LIN {X 0,Y 240.395,Z 425.258,A -85,B 0,C 180,E1 -19814.358,E2 -19814.358} C_VEL
LIN {X 0,Y 237.821,Z 422.9,A -85,B 0,C 180,E1 -19816.141,E2 -19816.141} C_VEL
LIN {X 0,Y 236.639,Z 420.217,A -85,B 0,C 180,E1 -19817.343,E2 -19817.343} C_VEL
LIN {X 0,Y 236.604,Z 420.167,A -85,B 0,C 180,E1 -19820.883,E2 -19820.883} C_VEL
LIN {X 0,Y 236.627,Z 420.436,A -85,B 0,C 180,E1 -19824.572,E2 -19824.572} C_VEL
LIN {X 0,Y 236.725,Z 421.066,A -85,B 0,C 180,E1 -19828.362,E2 -19828.362} C_VEL
LIN {X 0,Y 236.86,Z 422.112,A -85,B 0,C 180,E1 -19832.284,E2 -19832.284} C_VEL
LIN {X 0,Y 237.127,Z 423.615,A -85,B 0,C 180,E1 -19836.355,E2 -19836.355} C_VEL
LIN {X 0,Y 237.519,Z 425.71,A -85,B 0,C 180,E1 -19840.616,E2 -19840.616} C_VEL
LIN {X 0,Y 237.77,Z 427.097,A -85,B 0,C 180,E1 -19843.015,E2 -19843.015} C_VEL
LIN {X 0,Y 237.655,Z 428.197,A -85,B 0,C 180,E1 -19843.759,E2 -19843.759} C_VEL
LIN {X 0,Y 237.217,Z 431.036,A -85,B 0,C 180,E1 -19844.653,E2 -19844.653} C_VEL
LIN {X 0,Y 236.854,Z 438.007,A -85,B 0,C 180,E1 -19846.253,E2 -19846.253} C_VEL
LIN {X 0,Y 237.602,Z 440.293,A -85,B 0,C 180,E1 -19847.045,E2 -19847.045} C_VEL
LIN {X 0,Y 238.71,Z 442.196,A -85,B 0,C 180,E1 -19847.865,E2 -19847.865} C_VEL
LIN {X 0,Y 241.116,Z 447.739,A -85,B 0,C 180,E1 -19849.805,E2 -19849.805} C_VEL
LIN {X 0,Y 243.272,Z 454.639,A -85,B 0,C 180,E1 -19851.771,E2 -19851.771} C_VEL
LIN {X 0,Y 245.138,Z 466.004,A -85,B 0,C 180,E1 -19854.44,E2 -19854.44} C_VEL
LIN {X 0,Y 245.966,Z 476.957,A -85,B 0,C 180,E1 -19856.903,E2 -19856.903} C_VEL
LIN {X 0,Y 245.658,Z 486.508,A -85,B 0,C 180,E1 -19859.013,E2 -19859.013} C_VEL
LIN {X 0,Y 244.271,Z 496.15,A -85,B 0,C 180,E1 -19861.197,E2 -19861.197} C_VEL
LIN {X 0,Y 242.996,Z 501.368,A -85,B 0,C 180,E1 -19862.443,E2 -19862.443} C_VEL
LIN {X 0,Y 239.073,Z 510.716,A -85,B 0,C 180,E1 -19864.778,E2 -19864.778} C_VEL
LIN {X 0,Y 235.521,Z 518.441,A -85,B 0,C 180,E1 -19867.182,E2 -19867.182} C_VEL
LIN {X 0,Y 232.602,Z 524.845,A -85,B 0,C 180,E1 -19869.702,E2 -19869.702} C_VEL
LIN {X 0,Y 230.441,Z 529.963,A -85,B 0,C 180,E1 -19872.25,E2 -19872.25} C_VEL
LIN {X 0,Y 227.887,Z 535.233,A -85,B 0,C 180,E1 -19875.724,E2 -19875.724} C_VEL
LIN {X 0,Y 227.074,Z 537.27,A -85,B 0,C 180,E1 -19877.495,E2 -19877.495} C_VEL
LIN {X 0,Y 226.494,Z 538.88,A -85,B 0,C 180,E1 -19879.277,E2 -19879.277} C_VEL
LIN {X 0,Y 225.828,Z 540.91,A -85,B 0,C 180,E1 -19882.856,E2 -19882.856} C_VEL
LIN {X 0,Y 225.781,Z 541.415,A -85,B 0,C 180,E1 -19884.939,E2 -19884.939} C_VEL
LIN {X 0,Y 225.916,Z 541.064,A -85,B 0,C 180,E1 -19888.224,E2 -19888.224} C_VEL
LIN {X 0,Y 226.064,Z 540.289,A -85,B 0,C 180,E1 -19890.007,E2 -19890.007} C_VEL
LIN {X 0,Y 225.977,Z 539.082,A -85,B 0,C 180,E1 -19891.789,E2 -19891.789} C_VEL
LIN {X 0,Y 226.017,Z 536.428,A -85,B 0,C 180,E1 -19894.465,E2 -19894.465} C_VEL
LIN {X 0,Y 226.071,Z 532.684,A -85,B 0,C 180,E1 -19897.15,E2 -19897.15} C_VEL
LIN {X 0,Y 226.387,Z 527.772,A -85,B 0,C 180,E1 -19899.837,E2 -19899.837} C_VEL
LIN {X 0,Y 227.006,Z 521.552,A -85,B 0,C 180,E1 -19902.523,E2 -19902.523} C_VEL
LIN {X 0,Y 228.165,Z 513.778,A -85,B 0,C 180,E1 -19905.184,E2 -19905.184} C_VEL
LIN {X 0,Y 229.487,Z 504.066,A -85,B 0,C 180,E1 -19907.839,E2 -19907.839} C_VEL
LIN {X 0,Y 231.269,Z 494.144,A -85,B 0,C 180,E1 -19909.997,E2 -19909.997} C_VEL
LIN {X 0,Y 232.165,Z 486.97,A -85,B 0,C 180,E1 -19911.307,E2 -19911.307} C_VEL
LIN {X 0,Y 231.576,Z 476.41,A -85,B 0,C 180,E1 -19913.007,E2 -19913.007} C_VEL
LIN {X 0,Y 230.692,Z 464.985,A -85,B 0,C 180,E1 -19914.519,E2 -19914.519} C_VEL
LIN {X 0,Y 229.348,Z 451.694,A -85,B 0,C 180,E1 -19915.93,E2 -19915.93} C_VEL
LIN {X 0,Y 227.728,Z 438.212,A -85,B 0,C 180,E1 -19917.017,E2 -19917.017} C_VEL
LIN {X 0,Y 227.566,Z 436.511,A -85,B 0,C 180,E1 -19917.125,E2 -19917.125} C_VEL
LIN {X 0,Y 228.588,Z 431.326,A -85,B 0,C 180,E1 -19921.518,E2 -19921.518} C_VEL
LIN {X 0,Y 229.756,Z 426.613,A -85,B 0,C 180,E1 -19925.541,E2 -19925.541} C_VEL
LIN {X 0,Y 230.008,Z 424.188,A -85,B 0,C 180,E1 -19927.676,E2 -19927.676} C_VEL
LIN {X 0,Y 229.5,Z 420.39,A -85,B 0,C 180,E1 -19931.183,E2 -19931.183} C_VEL
LIN {X 0,Y 228.708,Z 416.42,A -85,B 0,C 180,E1 -19935.025,E2 -19935.025} C_VEL
LIN {X 0,Y 227.915,Z 412.095,A -85,B 0,C 180,E1 -19939.495,E2 -19939.495} C_VEL
LIN {X 0,Y 227.883,Z 412.095,A -85,B 0,C 180,E1 -19944.127,E2 -19944.127} C_VEL
LIN {X 0,Y 227.875,Z 412.098,A -85,B 0,C 180,E1 -19948.377,E2 -19948.377} C_VEL
LIN {X 0,Y 227.874,Z 412.097,A -85,B 0,C 180,E1 -19952.442,E2 -19952.442} C_VEL
LIN {X 0,Y 227.909,Z 412.094,A -85,B 0,C 180,E1 -19956.365,E2 -19956.365} C_VEL
LIN {X 0,Y 227.916,Z 412.092,A -85,B 0,C 180,E1 -19960.171,E2 -19960.171} C_VEL
LIN {X 0,Y 228.037,Z 412.077,A -85,B 0,C 180,E1 -19963.895,E2 -19963.895} C_VEL
LIN {X 0,Y 228.072,Z 412.073,A -85,B 0,C 180,E1 -19967.542,E2 -19967.542} C_VEL
LIN {X 0,Y 228.276,Z 412.05,A -85,B 0,C 180,E1 -19971.143,E2 -19971.143} C_VEL
LIN {X 0,Y 228.329,Z 412.044,A -85,B 0,C 180,E1 -19972.926,E2 -19972.926} C_VEL
LIN {X 0,Y 228.568,Z 412.009,A -85,B 0,C 180,E1 -19978.236,E2 -19978.236} C_VEL
LIN {X 0,Y 228.556,Z 412.013,A -85,B 0,C 180,E1 -19981.761,E2 -19981.761} C_VEL
LIN {X 0,Y 228.315,Z 412.044,A -85,B 0,C 180,E1 -19987.071,E2 -19987.071} C_VEL
LIN {X 0,Y 228.157,Z 412.065,A -85,B 0,C 180,E1 -19990.649,E2 -19990.649} C_VEL
LIN {X 0,Y 228.047,Z 412.076,A -85,B 0,C 180,E1 -19994.272,E2 -19994.272} C_VEL
LIN {X 0,Y 227.945,Z 412.089,A -85,B 0,C 180,E1 -19997.956,E2 -19997.956} C_VEL
LIN {X 0,Y 227.914,Z 412.093,A -85,B 0,C 180,E1 -20002.306,E2 -20002.306} C_VEL
LIN {X 0,Y 227.954,Z 412.091,A -85,B 0,C 180,E1 -20006.597,E2 -20006.597} C_VEL
LIN {X 0,Y 227.89,Z 412.097,A -85,B 0,C 180,E1 -20010.278,E2 -20010.278} C_VEL
LIN {X 0,Y 227.889,Z 412.095,A -85,B 0,C 180,E1 -20013.716,E2 -20013.716} C_VEL
LIN {X 0,Y 227.855,Z 412.101,A -85,B 0,C 180,E1 -20018.087,E2 -20018.087} C_VEL
LIN {X 0,Y 227.815,Z 412.108,A -85,B 0,C 180,E1 -20022.739,E2 -20022.739} C_VEL
LIN {X 0,Y 227.811,Z 412.104,A -85,B 0,C 180,E1 -20027.25,E2 -20027.25} C_VEL
LIN {X 0,Y 227.85,Z 412.101,A -85,B 0,C 180,E1 -20031.903,E2 -20031.903} C_VEL
LIN {X 0,Y 227.885,Z 412.098,A -85,B 0,C 180,E1 -20036.372,E2 -20036.372} C_VEL
LIN {X 0,Y 227.923,Z 412.096,A -85,B 0,C 180,E1 -20040.432,E2 -20040.432} C_VEL
LIN {X 0,Y 227.932,Z 412.091,A -85,B 0,C 180,E1 -20044.42,E2 -20044.42} C_VEL
LIN {X 0,Y 227.965,Z 412.09,A -85,B 0,C 180,E1 -20048.281,E2 -20048.281} C_VEL
LIN {X 0,Y 228.035,Z 412.076,A -85,B 0,C 180,E1 -20052.82,E2 -20052.82} C_VEL
LIN {X 0,Y 228.071,Z 412.074,A -85,B 0,C 180,E1 -20057.537,E2 -20057.537} C_VEL
LIN {X 0,Y 228.265,Z 412.047,A -85,B 0,C 180,E1 -20061.138,E2 -20061.138} C_VEL
LIN {X 0,Y 228.32,Z 412.041,A -85,B 0,C 180,E1 -20062.921,E2 -20062.921} C_VEL
LIN {X 0,Y 228.548,Z 412.016,A -85,B 0,C 180,E1 -20068.231,E2 -20068.231} C_VEL
LIN {X 0,Y 228.548,Z 412.013,A -85,B 0,C 180,E1 -20071.756,E2 -20071.756} C_VEL
LIN {X 0,Y 228.348,Z 412.038,A -85,B 0,C 180,E1 -20077.065,E2 -20077.065} C_VEL
LIN {X 0,Y 228.16,Z 412.063,A -85,B 0,C 180,E1 -20080.644,E2 -20080.644} C_VEL
LIN {X 0,Y 228.044,Z 412.077,A -85,B 0,C 180,E1 -20086.096,E2 -20086.096} C_VEL
LIN {X 0,Y 227.921,Z 412.094,A -85,B 0,C 180,E1 -20089.82,E2 -20089.82} C_VEL
LIN {X 0,Y 227.835,Z 412.104,A -85,B 0,C 180,E1 -20093.633,E2 -20093.633} C_VEL
LIN {X 0,Y 227.596,Z 412.134,A -85,B 0,C 180,E1 -20097.585,E2 -20097.585} C_VEL
LIN {X 0,Y 227.351,Z 412.166,A -85,B 0,C 180,E1 -20100.058,E2 -20100.058} C_VEL
LIN {X 0,Y 226.798,Z 412.354,A -85,B 0,C 180,E1 -20105.037,E2 -20105.037} C_VEL
LIN {X 0,Y 229.937,Z 425.401,A -85,B 0,C 180,E1 -20106.238,E2 -20106.238} C_VEL
LIN {X 0,Y 232.669,Z 438.268,A -85,B 0,C 180,E1 -20107.723,E2 -20107.723} C_VEL
LIN {X 0,Y 234.88,Z 450.436,A -85,B 0,C 180,E1 -20109.443,E2 -20109.443} C_VEL
LIN {X 0,Y 233.284,Z 461.497,A -85,B 0,C 180,E1 -20111.138,E2 -20111.138} C_VEL
LIN {X 0,Y 231.588,Z 472.576,A -85,B 0,C 180,E1 -20113.256,E2 -20113.256} C_VEL
LIN {X 0,Y 229.953,Z 482.534,A -85,B 0,C 180,E1 -20115.646,E2 -20115.646} C_VEL
LIN {X 0,Y 228.635,Z 490.664,A -85,B 0,C 180,E1 -20118.045,E2 -20118.045} C_VEL
LIN {X 0,Y 227.625,Z 497.485,A -85,B 0,C 180,E1 -20120.511,E2 -20120.511} C_VEL
LIN {X 0,Y 226.877,Z 502.686,A -85,B 0,C 180,E1 -20122.813,E2 -20122.813} C_VEL
LIN {X 0,Y 226.214,Z 508.373,A -85,B 0,C 180,E1 -20126,E2 -20126} C_VEL
LIN {X 0,Y 225.792,Z 512.402,A -85,B 0,C 180,E1 -20129.1,E2 -20129.1} C_VEL
LIN {X 0,Y 225.652,Z 515.079,A -85,B 0,C 180,E1 -20132.151,E2 -20132.151} C_VEL
LIN {X 0,Y 225.873,Z 516.315,A -85,B 0,C 180,E1 -20134.447,E2 -20134.447} C_VEL
LIN {X 0,Y 226.125,Z 516.805,A -85,B 0,C 180,E1 -20136.171,E2 -20136.171} C_VEL
LIN {X 0,Y 226.703,Z 516.93,A -85,B 0,C 180,E1 -20138.417,E2 -20138.417} C_VEL
LIN {X 0,Y 227.291,Z 516.575,A -85,B 0,C 180,E1 -20140.117,E2 -20140.117} C_VEL
LIN {X 0,Y 228.369,Z 515.473,A -85,B 0,C 180,E1 -20142.529,E2 -20142.529} C_VEL
LIN {X 0,Y 230.39,Z 512.669,A -85,B 0,C 180,E1 -20145.877,E2 -20145.877} C_VEL
LIN {X 0,Y 232.621,Z 509.086,A -85,B 0,C 180,E1 -20148.676,E2 -20148.676} C_VEL
LIN {X 0,Y 235.316,Z 504.302,A -85,B 0,C 180,E1 -20151.413,E2 -20151.413} C_VEL
LIN {X 0,Y 238.496,Z 498.196,A -85,B 0,C 180,E1 -20154.082,E2 -20154.082} C_VEL
LIN {X 0,Y 242.228,Z 490.525,A -85,B 0,C 180,E1 -20156.675,E2 -20156.675} C_VEL
LIN {X 0,Y 245.987,Z 481.918,A -85,B 0,C 180,E1 -20158.951,E2 -20158.951} C_VEL
LIN {X 0,Y 249.82,Z 472.11,A -85,B 0,C 180,E1 -20161.009,E2 -20161.009} C_VEL
LIN {X 0,Y 250.157,Z 471.048,A -85,B 0,C 180,E1 -20161.209,E2 -20161.209} C_VEL
LIN {X 0,Y 250.135,Z 467.345,A -85,B 0,C 180,E1 -20162.198,E2 -20162.198} C_VEL
LIN {X 0,Y 248.511,Z 456.289,A -85,B 0,C 180,E1 -20165.275,E2 -20165.275} C_VEL
LIN {X 0,Y 247.07,Z 450.957,A -85,B 0,C 180,E1 -20166.903,E2 -20166.903} C_VEL
LIN {X 0,Y 243.973,Z 443.043,A -85,B 0,C 180,E1 -20169.59,E2 -20169.59} C_VEL
LIN {X 0,Y 240.468,Z 436.403,A -85,B 0,C 180,E1 -20172.332,E2 -20172.332} C_VEL
LIN {X 0,Y 238.036,Z 432.974,A -85,B 0,C 180,E1 -20174.155,E2 -20174.155} C_VEL
LIN {X 0,Y 237.523,Z 431.74,A -85,B 0,C 180,E1 -20174.656,E2 -20174.656} C_VEL
LIN {X 0,Y 234.864,Z 428.845,A -85,B 0,C 180,E1 -20176.781,E2 -20176.781} C_VEL
LIN {X 0,Y 233.933,Z 426.768,A -85,B 0,C 180,E1 -20177.799,E2 -20177.799} C_VEL
LIN {X 0,Y 231.195,Z 424.804,A -85,B 0,C 180,E1 -20180.37,E2 -20180.37} C_VEL
LIN {X 0,Y 229.79,Z 422.242,A -85,B 0,C 180,E1 -20182.459,E2 -20182.459} C_VEL
LIN {X 0,Y 229.723,Z 421.918,A -85,B 0,C 180,E1 -20182.783,E2 -20182.783} C_VEL
LIN {X 0,Y 229.799,Z 422.557,A -85,B 0,C 180,E1 -20187.53,E2 -20187.53} C_VEL
LIN {X 0,Y 229.913,Z 423.479,A -85,B 0,C 180,E1 -20191.311,E2 -20191.311} C_VEL
LIN {X 0,Y 230.131,Z 424.91,A -85,B 0,C 180,E1 -20195.469,E2 -20195.469} C_VEL
LIN {X 0,Y 230.549,Z 426.955,A -85,B 0,C 180,E1 -20199.983,E2 -20199.983} C_VEL
LIN {X 0,Y 230.78,Z 427.896,A -85,B 0,C 180,E1 -20200.528,E2 -20200.528} C_VEL
LIN {X 0,Y 232.478,Z 431.639,A -85,B 0,C 180,E1 -20202.592,E2 -20202.592} C_VEL
LIN {X 0,Y 235.284,Z 435.262,A -85,B 0,C 180,E1 -20204.981,E2 -20204.981} C_VEL
LIN {X 0,Y 236.767,Z 439.078,A -85,B 0,C 180,E1 -20206.443,E2 -20206.443} C_VEL
LIN {X 0,Y 237.602,Z 440.293,A -85,B 0,C 180,E1 -20207.045,E2 -20207.045} C_VEL
LIN {X 0,Y 238.57,Z 442.303,A -85,B 0,C 180,E1 -20207.821,E2 -20207.821} C_VEL
LIN {X 0,Y 239.346,Z 446.289,A -85,B 0,C 180,E1 -20208.853,E2 -20208.853} C_VEL
LIN {X 0,Y 239.528,Z 450.901,A -85,B 0,C 180,E1 -20209.76,E2 -20209.76} C_VEL
LIN {X 0,Y 239.223,Z 460.716,A -85,B 0,C 180,E1 -20211.548,E2 -20211.548} C_VEL
LIN {X 0,Y 239.322,Z 463.717,A -85,B 0,C 180,E1 -20212.216,E2 -20212.216} C_VEL
LIN {X 0,Y 240.312,Z 474.933,A -85,B 0,C 180,E1 -20214.974,E2 -20214.974} C_VEL
LIN {X 0,Y 240.144,Z 484.437,A -85,B 0,C 180,E1 -20217.228,E2 -20217.228} C_VEL
LIN {X 0,Y 238.986,Z 493.867,A -85,B 0,C 180,E1 -20219.474,E2 -20219.474} C_VEL
LIN {X 0,Y 236.802,Z 502.601,A -85,B 0,C 180,E1 -20221.658,E2 -20221.658} C_VEL
LIN {X 0,Y 232.733,Z 511.624,A -85,B 0,C 180,E1 -20224.04,E2 -20224.04} C_VEL
LIN {X 0,Y 228.479,Z 520.166,A -85,B 0,C 180,E1 -20226.917,E2 -20226.917} C_VEL
LIN {X 0,Y 225.135,Z 526.962,A -85,B 0,C 180,E1 -20229.924,E2 -20229.924} C_VEL
LIN {X 0,Y 222.947,Z 531.621,A -85,B 0,C 180,E1 -20232.582,E2 -20232.582} C_VEL
LIN {X 0,Y 221.001,Z 535.271,A -85,B 0,C 180,E1 -20235.269,E2 -20235.269} C_VEL
LIN {X 0,Y 219.472,Z 538.676,A -85,B 0,C 180,E1 -20238.93,E2 -20238.93} C_VEL
LIN {X 0,Y 218.777,Z 540.58,A -85,B 0,C 180,E1 -20242.624,E2 -20242.624} C_VEL
LIN {X 0,Y 218.712,Z 540.966,A -85,B 0,C 180,E1 -20244.979,E2 -20244.979} C_VEL
LIN {X 0,Y 218.843,Z 540.48,A -85,B 0,C 180,E1 -20248.166,E2 -20248.166} C_VEL
LIN {X 0,Y 218.987,Z 539.652,A -85,B 0,C 180,E1 -20250.007,E2 -20250.007} C_VEL
LIN {X 0,Y 218.908,Z 538.39,A -85,B 0,C 180,E1 -20251.846,E2 -20251.846} C_VEL
LIN {X 0,Y 218.947,Z 535.215,A -85,B 0,C 180,E1 -20254.934,E2 -20254.934} C_VEL
LIN {X 0,Y 219.016,Z 531.734,A -85,B 0,C 180,E1 -20257.381,E2 -20257.381} C_VEL
LIN {X 0,Y 219.452,Z 525.674,A -85,B 0,C 180,E1 -20260.618,E2 -20260.618} C_VEL
LIN {X 0,Y 220.231,Z 519.02,A -85,B 0,C 180,E1 -20263.384,E2 -20263.384} C_VEL
LIN {X 0,Y 221.484,Z 510.777,A -85,B 0,C 180,E1 -20266.126,E2 -20266.126} C_VEL
LIN {X 0,Y 222.959,Z 501.162,A -85,B 0,C 180,E1 -20268.665,E2 -20268.665} C_VEL
LIN {X 0,Y 224.704,Z 490.884,A -85,B 0,C 180,E1 -20270.847,E2 -20270.847} C_VEL
LIN {X 0,Y 225.12,Z 487.183,A -85,B 0,C 180,E1 -20271.526,E2 -20271.526} C_VEL
LIN {X 0,Y 224.548,Z 476.756,A -85,B 0,C 180,E1 -20273.281,E2 -20273.281} C_VEL
LIN {X 0,Y 223.579,Z 464.048,A -85,B 0,C 180,E1 -20275.029,E2 -20275.029} C_VEL
LIN {X 0,Y 222.258,Z 450.417,A -85,B 0,C 180,E1 -20276.512,E2 -20276.512} C_VEL
LIN {X 0,Y 220.574,Z 436.104,A -85,B 0,C 180,E1 -20277.696,E2 -20277.696} C_VEL
LIN {X 0,Y 221.775,Z 430.52,A -85,B 0,C 180,E1 -20282.604,E2 -20282.604} C_VEL
LIN {X 0,Y 222.721,Z 427.001,A -85,B 0,C 180,E1 -20285.722,E2 -20285.722} C_VEL
LIN {X 0,Y 222.925,Z 424.531,A -85,B 0,C 180,E1 -20287.984,E2 -20287.984} C_VEL
LIN {X 0,Y 222.357,Z 420.746,A -85,B 0,C 180,E1 -20291.593,E2 -20291.593} C_VEL
LIN {X 0,Y 221.545,Z 416.633,A -85,B 0,C 180,E1 -20295.739,E2 -20295.739} C_VEL
LIN {X 0,Y 220.868,Z 412.971,A -85,B 0,C 180,E1 -20299.798,E2 -20299.798} C_VEL
LIN {X 0,Y 220.844,Z 412.975,A -85,B 0,C 180,E1 -20302.795,E2 -20302.795} C_VEL
LIN {X 0,Y 220.831,Z 412.978,A -85,B 0,C 180,E1 -20307.245,E2 -20307.245} C_VEL
LIN {X 0,Y 220.823,Z 412.976,A -85,B 0,C 180,E1 -20311.483,E2 -20311.483} C_VEL
LIN {X 0,Y 220.864,Z 412.972,A -85,B 0,C 180,E1 -20315.563,E2 -20315.563} C_VEL
LIN {X 0,Y 220.873,Z 412.97,A -85,B 0,C 180,E1 -20319.51,E2 -20319.51} C_VEL
LIN {X 0,Y 220.995,Z 412.956,A -85,B 0,C 180,E1 -20323.367,E2 -20323.367} C_VEL
LIN {X 0,Y 221.08,Z 412.945,A -85,B 0,C 180,E1 -20329.003,E2 -20329.003} C_VEL
LIN {X 0,Y 221.265,Z 412.922,A -85,B 0,C 180,E1 -20332.699,E2 -20332.699} C_VEL
LIN {X 0,Y 221.525,Z 412.886,A -85,B 0,C 180,E1 -20338.18,E2 -20338.18} C_VEL
LIN {X 0,Y 221.489,Z 412.893,A -85,B 0,C 180,E1 -20341.817,E2 -20341.817} C_VEL
LIN {X 0,Y 221.253,Z 412.922,A -85,B 0,C 180,E1 -20347.298,E2 -20347.298} C_VEL
LIN {X 0,Y 221.078,Z 412.947,A -85,B 0,C 180,E1 -20350.994,E2 -20350.994} C_VEL
LIN {X 0,Y 220.992,Z 412.956,A -85,B 0,C 180,E1 -20356.63,E2 -20356.63} C_VEL
LIN {X 0,Y 220.866,Z 412.973,A -85,B 0,C 180,E1 -20360.487,E2 -20360.487} C_VEL
LIN {X 0,Y 220.874,Z 412.969,A -85,B 0,C 180,E1 -20364.432,E2 -20364.432} C_VEL
LIN {X 0,Y 220.827,Z 412.979,A -85,B 0,C 180,E1 -20368.513,E2 -20368.513} C_VEL
LIN {X 0,Y 220.825,Z 412.977,A -85,B 0,C 180,E1 -20372.753,E2 -20372.753} C_VEL
LIN {X 0,Y 220.821,Z 412.977,A -85,B 0,C 180,E1 -20377.273,E2 -20377.273} C_VEL
LIN {X 0,Y 220.805,Z 412.978,A -85,B 0,C 180,E1 -20380.183,E2 -20380.183} C_VEL
LIN {X 0,Y 220.776,Z 412.986,A -85,B 0,C 180,E1 -20384.451,E2 -20384.451} C_VEL
LIN {X 0,Y 220.769,Z 412.982,A -85,B 0,C 180,E1 -20388.04,E2 -20388.04} C_VEL
LIN {X 0,Y 220.832,Z 412.977,A -85,B 0,C 180,E1 -20392.787,E2 -20392.787} C_VEL
LIN {X 0,Y 220.823,Z 412.974,A -85,B 0,C 180,E1 -20397.238,E2 -20397.238} C_VEL
LIN {X 0,Y 220.84,Z 412.974,A -85,B 0,C 180,E1 -20401.48,E2 -20401.48} C_VEL
LIN {X 0,Y 220.871,Z 412.967,A -85,B 0,C 180,E1 -20405.559,E2 -20405.559} C_VEL
LIN {X 0,Y 220.895,Z 412.968,A -85,B 0,C 180,E1 -20409.508,E2 -20409.508} C_VEL
LIN {X 0,Y 221.017,Z 412.949,A -85,B 0,C 180,E1 -20413.364,E2 -20413.364} C_VEL
LIN {X 0,Y 221.08,Z 412.944,A -85,B 0,C 180,E1 -20418.998,E2 -20418.998} C_VEL
LIN {X 0,Y 221.256,Z 412.922,A -85,B 0,C 180,E1 -20422.694,E2 -20422.694} C_VEL
LIN {X 0,Y 221.506,Z 412.894,A -85,B 0,C 180,E1 -20428.175,E2 -20428.175} C_VEL
LIN {X 0,Y 221.506,Z 412.891,A -85,B 0,C 180,E1 -20431.811,E2 -20431.811} C_VEL
LIN {X 0,Y 221.301,Z 412.916,A -85,B 0,C 180,E1 -20437.291,E2 -20437.291} C_VEL
LIN {X 0,Y 221.106,Z 412.941,A -85,B 0,C 180,E1 -20440.987,E2 -20440.987} C_VEL
LIN {X 0,Y 221.002,Z 412.951,A -85,B 0,C 180,E1 -20446.623,E2 -20446.623} C_VEL
LIN {X 0,Y 220.869,Z 412.972,A -85,B 0,C 180,E1 -20450.481,E2 -20450.481} C_VEL
LIN {X 0,Y 220.746,Z 412.987,A -85,B 0,C 180,E1 -20454.441,E2 -20454.441} C_VEL
LIN {X 0,Y 220.632,Z 413,A -85,B 0,C 180,E1 -20456.89,E2 -20456.89} C_VEL
LIN {X 0,Y 220.19,Z 413.056,A -85,B 0,C 180,E1 -20460.701,E2 -20460.701} C_VEL
LIN {X 0,Y 219.774,Z 413.214,A -85,B 0,C 180,E1 -20464.516,E2 -20464.516} C_VEL
LIN {X 0,Y 222.803,Z 425.42,A -85,B 0,C 180,E1 -20465.692,E2 -20465.692} C_VEL
LIN {X 0,Y 225.456,Z 437.626,A -85,B 0,C 180,E1 -20467.145,E2 -20467.145} C_VEL
LIN {X 0,Y 227.578,Z 449.266,A -85,B 0,C 180,E1 -20468.805,E2 -20468.805} C_VEL
LIN {X 0,Y 227.774,Z 452.159,A -85,B 0,C 180,E1 -20469.257,E2 -20469.257} C_VEL
LIN {X 0,Y 226.028,Z 463.808,A -85,B 0,C 180,E1 -20471.147,E2 -20471.147} C_VEL
LIN {X 0,Y 224.387,Z 474.089,A -85,B 0,C 180,E1 -20473.247,E2 -20473.247} C_VEL
LIN {X 0,Y 222.894,Z 482.923,A -85,B 0,C 180,E1 -20475.451,E2 -20475.451} C_VEL
LIN {X 0,Y 221.45,Z 491.907,A -85,B 0,C 180,E1 -20478.208,E2 -20478.208} C_VEL
LIN {X 0,Y 220.369,Z 499.042,A -85,B 0,C 180,E1 -20480.962,E2 -20480.962} C_VEL
LIN {X 0,Y 219.524,Z 505.151,A -85,B 0,C 180,E1 -20483.94,E2 -20483.94} C_VEL
LIN {X 0,Y 218.983,Z 509.905,A -85,B 0,C 180,E1 -20486.937,E2 -20486.937} C_VEL
LIN {X 0,Y 218.602,Z 513.697,A -85,B 0,C 180,E1 -20490.215,E2 -20490.215} C_VEL
LIN {X 0,Y 218.747,Z 516.415,A -85,B 0,C 180,E1 -20494.086,E2 -20494.086} C_VEL
LIN {X 0,Y 219.313,Z 517.384,A -85,B 0,C 180,E1 -20497.386,E2 -20497.386} C_VEL
LIN {X 0,Y 219.935,Z 517.322,A -85,B 0,C 180,E1 -20499.423,E2 -20499.423} C_VEL
LIN {X 0,Y 221.185,Z 516.407,A -85,B 0,C 180,E1 -20502.379,E2 -20502.379} C_VEL
LIN {X 0,Y 222.938,Z 514.387,A -85,B 0,C 180,E1 -20505.394,E2 -20505.394} C_VEL
LIN {X 0,Y 225.125,Z 511.316,A -85,B 0,C 180,E1 -20508.294,E2 -20508.294} C_VEL
LIN {X 0,Y 227.784,Z 507.111,A -85,B 0,C 180,E1 -20511.127,E2 -20511.127} C_VEL
LIN {X 0,Y 231.006,Z 501.658,A -85,B 0,C 180,E1 -20513.889,E2 -20513.889} C_VEL
LIN {X 0,Y 234.8,Z 494.716,A -85,B 0,C 180,E1 -20516.57,E2 -20516.57} C_VEL
LIN {X 0,Y 238.944,Z 486.035,A -85,B 0,C 180,E1 -20519.166,E2 -20519.166} C_VEL
LIN {X 0,Y 243.238,Z 476.27,A -85,B 0,C 180,E1 -20521.45,E2 -20521.45} C_VEL
LIN {X 0,Y 244.417,Z 473.241,A -85,B 0,C 180,E1 -20522.061,E2 -20522.061} C_VEL
LIN {X 0,Y 244.125,Z 467.412,A -85,B 0,C 180,E1 -20523.791,E2 -20523.791} C_VEL
LIN {X 0,Y 243.271,Z 459.836,A -85,B 0,C 180,E1 -20526.054,E2 -20526.054} C_VEL
LIN {X 0,Y 241.347,Z 452.92,A -85,B 0,C 180,E1 -20528.373,E2 -20528.373} C_VEL
LIN {X 0,Y 238.964,Z 446.64,A -85,B 0,C 180,E1 -20530.786,E2 -20530.786} C_VEL
LIN {X 0,Y 236.294,Z 441.604,A -85,B 0,C 180,E1 -20533.159,E2 -20533.159} C_VEL
LIN {X 0,Y 234.338,Z 437.991,A -85,B 0,C 180,E1 -20535.021,E2 -20535.021} C_VEL
LIN {X 0,Y 232.422,Z 435.783,A -85,B 0,C 180,E1 -20536.696,E2 -20536.696} C_VEL
LIN {X 0,Y 231.56,Z 434.156,A -85,B 0,C 180,E1 -20537.67,E2 -20537.67} C_VEL
LIN {X 0,Y 227.769,Z 429.425,A -85,B 0,C 180,E1 -20542.441,E2 -20542.441} C_VEL
LIN {X 0,Y 227.494,Z 428.674,A -85,B 0,C 180,E1 -20543.025,E2 -20543.025} C_VEL
LIN {X 0,Y 225.122,Z 427.997,A -85,B 0,C 180,E1 -20547.924,E2 -20547.924} C_VEL
LIN {X 0,Y 224.813,Z 428.537,A -85,B 0,C 180,E1 -20551.642,E2 -20551.642} C_VEL
LIN {X 0,Y 225.522,Z 430.166,A -85,B 0,C 180,E1 -20555.049,E2 -20555.049} C_VEL
LIN {X 0,Y 228.23,Z 433.772,A -85,B 0,C 180,E1 -20559.764,E2 -20559.764} C_VEL
LIN {X 0,Y 229.134,Z 436.616,A -85,B 0,C 180,E1 -20561.26,E2 -20561.26} C_VEL
LIN {X 0,Y 231.961,Z 440.862,A -85,B 0,C 180,E1 -20564.177,E2 -20564.177} C_VEL
LIN {X 0,Y 233.896,Z 445.696,A -85,B 0,C 180,E1 -20566.294,E2 -20566.294} C_VEL
LIN {X 0,Y 234.925,Z 447.325,A -85,B 0,C 180,E1 -20567.099,E2 -20567.099} C_VEL
LIN {X 0,Y 237.157,Z 453.445,A -85,B 0,C 180,E1 -20569.321,E2 -20569.321} C_VEL
LIN {X 0,Y 238.707,Z 459.159,A -85,B 0,C 180,E1 -20571.042,E2 -20571.042} C_VEL
LIN {X 0,Y 239.322,Z 463.717,A -85,B 0,C 180,E1 -20572.216,E2 -20572.216} C_VEL
LIN {X 0,Y 239.258,Z 468.21,A -85,B 0,C 180,E1 -20573.157,E2 -20573.157} C_VEL
LIN {X 0,Y 238.343,Z 473.068,A -85,B 0,C 180,E1 -20573.977,E2 -20573.977} C_VEL
LIN {X 0,Y 235.547,Z 482.684,A -85,B 0,C 180,E1 -20575.571,E2 -20575.571} C_VEL
LIN {X 0,Y 234.192,Z 488.536,A -85,B 0,C 180,E1 -20576.833,E2 -20576.833} C_VEL
LIN {X 0,Y 232.649,Z 497.379,A -85,B 0,C 180,E1 -20579.108,E2 -20579.108} C_VEL
LIN {X 0,Y 230.661,Z 503.871,A -85,B 0,C 180,E1 -20580.832,E2 -20580.832} C_VEL
LIN {X 0,Y 226.435,Z 512.496,A -85,B 0,C 180,E1 -20583.262,E2 -20583.262} C_VEL
LIN {X 0,Y 222.566,Z 519.701,A -85,B 0,C 180,E1 -20585.772,E2 -20585.772} C_VEL
LIN {X 0,Y 219.075,Z 526.217,A -85,B 0,C 180,E1 -20588.694,E2 -20588.694} C_VEL
LIN {X 0,Y 216.181,Z 531.75,A -85,B 0,C 180,E1 -20592.018,E2 -20592.018} C_VEL
LIN {X 0,Y 214.135,Z 535.252,A -85,B 0,C 180,E1 -20594.785,E2 -20594.785} C_VEL
LIN {X 0,Y 212.461,Z 538.498,A -85,B 0,C 180,E1 -20598.56,E2 -20598.56} C_VEL
LIN {X 0,Y 212.005,Z 539.56,A -85,B 0,C 180,E1 -20600.467,E2 -20600.467} C_VEL
LIN {X 0,Y 211.627,Z 540.499,A -85,B 0,C 180,E1 -20604.289,E2 -20604.289} C_VEL
LIN {X 0,Y 211.676,Z 540.389,A -85,B 0,C 180,E1 -20606.2,E2 -20606.2} C_VEL
LIN {X 0,Y 211.772,Z 539.89,A -85,B 0,C 180,E1 -20608.105,E2 -20608.105} C_VEL
LIN {X 0,Y 211.912,Z 538.994,A -85,B 0,C 180,E1 -20610.007,E2 -20610.007} C_VEL
LIN {X 0,Y 211.841,Z 537.61,A -85,B 0,C 180,E1 -20611.908,E2 -20611.908} C_VEL
LIN {X 0,Y 211.904,Z 534.548,A -85,B 0,C 180,E1 -20614.9,E2 -20614.9} C_VEL
LIN {X 0,Y 211.988,Z 530.711,A -85,B 0,C 180,E1 -20617.627,E2 -20617.627} C_VEL
LIN {X 0,Y 212.443,Z 524.491,A -85,B 0,C 180,E1 -20620.972,E2 -20620.972} C_VEL
LIN {X 0,Y 213.316,Z 517.69,A -85,B 0,C 180,E1 -20623.826,E2 -20623.826} C_VEL
LIN {X 0,Y 214.374,Z 510.735,A -85,B 0,C 180,E1 -20626.187,E2 -20626.187} C_VEL
LIN {X 0,Y 215.647,Z 502.355,A -85,B 0,C 180,E1 -20628.534,E2 -20628.534} C_VEL
LIN {X 0,Y 217.461,Z 492.176,A -85,B 0,C 180,E1 -20630.831,E2 -20630.831} C_VEL
LIN {X 0,Y 218.072,Z 487.395,A -85,B 0,C 180,E1 -20631.76,E2 -20631.76} C_VEL
LIN {X 0,Y 217.432,Z 475.475,A -85,B 0,C 180,E1 -20633.837,E2 -20633.837} C_VEL
LIN {X 0,Y 216.434,Z 462.757,A -85,B 0,C 180,E1 -20635.619,E2 -20635.619} C_VEL
LIN {X 0,Y 215.163,Z 449.603,A -85,B 0,C 180,E1 -20637.088,E2 -20637.088} C_VEL
LIN {X 0,Y 213.596,Z 435.722,A -85,B 0,C 180,E1 -20638.281,E2 -20638.281} C_VEL
LIN {X 0,Y 214.712,Z 430.874,A -85,B 0,C 180,E1 -20642.696,E2 -20642.696} C_VEL
LIN {X 0,Y 215.665,Z 427.36,A -85,B 0,C 180,E1 -20645.921,E2 -20645.921} C_VEL
LIN {X 0,Y 215.803,Z 424.551,A -85,B 0,C 180,E1 -20648.59,E2 -20648.59} C_VEL
LIN {X 0,Y 215.366,Z 421.759,A -85,B 0,C 180,E1 -20651.359,E2 -20651.359} C_VEL
LIN {X 0,Y 214.345,Z 416.832,A -85,B 0,C 180,E1 -20656.482,E2 -20656.482} C_VEL
LIN {X 0,Y 213.826,Z 413.848,A -85,B 0,C 180,E1 -20659.923,E2 -20659.923} C_VEL
LIN {X 0,Y 213.785,Z 413.853,A -85,B 0,C 180,E1 -20665.28,E2 -20665.28} C_VEL
LIN {X 0,Y 213.788,Z 413.854,A -85,B 0,C 180,E1 -20668.739,E2 -20668.739} C_VEL
LIN {X 0,Y 213.808,Z 413.849,A -85,B 0,C 180,E1 -20672.599,E2 -20672.599} C_VEL
LIN {X 0,Y 213.82,Z 413.852,A -85,B 0,C 180,E1 -20676.987,E2 -20676.987} C_VEL
LIN {X 0,Y 213.904,Z 413.837,A -85,B 0,C 180,E1 -20682.799,E2 -20682.799} C_VEL
LIN {X 0,Y 213.951,Z 413.835,A -85,B 0,C 180,E1 -20686.705,E2 -20686.705} C_VEL
LIN {X 0,Y 214.155,Z 413.805,A -85,B 0,C 180,E1 -20690.554,E2 -20690.554} C_VEL
LIN {X 0,Y 214.106,Z 413.814,A -85,B 0,C 180,E1 -20694.347,E2 -20694.347} C_VEL
LIN {X 0,Y 214.459,Z 413.766,A -85,B 0,C 180,E1 -20698.12,E2 -20698.12} C_VEL
LIN {X 0,Y 214.554,Z 413.756,A -85,B 0,C 180,E1 -20699.998,E2 -20699.998} C_VEL
LIN {X 0,Y 214.426,Z 413.773,A -85,B 0,C 180,E1 -20701.877,E2 -20701.877} C_VEL
LIN {X 0,Y 214.194,Z 413.8,A -85,B 0,C 180,E1 -20707.54,E2 -20707.54} C_VEL
LIN {X 0,Y 214.009,Z 413.826,A -85,B 0,C 180,E1 -20711.362,E2 -20711.362} C_VEL
LIN {X 0,Y 213.913,Z 413.836,A -85,B 0,C 180,E1 -20715.237,E2 -20715.237} C_VEL
LIN {X 0,Y 213.811,Z 413.851,A -85,B 0,C 180,E1 -20719.188,E2 -20719.188} C_VEL
LIN {X 0,Y 213.812,Z 413.847,A -85,B 0,C 180,E1 -20723.229,E2 -20723.229} C_VEL
LIN {X 0,Y 213.826,Z 413.848,A -85,B 0,C 180,E1 -20727.436,E2 -20727.436} C_VEL
LIN {X 0,Y 213.772,Z 413.851,A -85,B 0,C 180,E1 -20731.735,E2 -20731.735} C_VEL
LIN {X 0,Y 213.756,Z 413.859,A -85,B 0,C 180,E1 -20736.284,E2 -20736.284} C_VEL
LIN {X 0,Y 213.721,Z 413.86,A -85,B 0,C 180,E1 -20741.121,E2 -20741.121} C_VEL
LIN {X 0,Y 213.713,Z 413.862,A -85,B 0,C 180,E1 -20743.674,E2 -20743.674} C_VEL
LIN {X 0,Y 213.712,Z 413.865,A -85,B 0,C 180,E1 -20746.34,E2 -20746.34} C_VEL
LIN {X 0,Y 213.717,Z 413.86,A -85,B 0,C 180,E1 -20749.14,E2 -20749.14} C_VEL
LIN {X 0,Y 213.751,Z 413.858,A -85,B 0,C 180,E1 -20753.706,E2 -20753.706} C_VEL
LIN {X 0,Y 213.786,Z 413.854,A -85,B 0,C 180,E1 -20758.725,E2 -20758.725} C_VEL
LIN {X 0,Y 213.831,Z 413.849,A -85,B 0,C 180,E1 -20762.597,E2 -20762.597} C_VEL
LIN {X 0,Y 213.855,Z 413.844,A -85,B 0,C 180,E1 -20766.946,E2 -20766.946} C_VEL
LIN {X 0,Y 213.945,Z 413.831,A -85,B 0,C 180,E1 -20772.797,E2 -20772.797} C_VEL
LIN {X 0,Y 213.952,Z 413.834,A -85,B 0,C 180,E1 -20776.7,E2 -20776.7} C_VEL
LIN {X 0,Y 214.139,Z 413.808,A -85,B 0,C 180,E1 -20780.548,E2 -20780.548} C_VEL
LIN {X 0,Y 214.096,Z 413.817,A -85,B 0,C 180,E1 -20784.342,E2 -20784.342} C_VEL
LIN {X 0,Y 214.439,Z 413.774,A -85,B 0,C 180,E1 -20788.115,E2 -20788.115} C_VEL
LIN {X 0,Y 214.543,Z 413.759,A -85,B 0,C 180,E1 -20789.993,E2 -20789.993} C_VEL
LIN {X 0,Y 214.439,Z 413.771,A -85,B 0,C 180,E1 -20791.871,E2 -20791.871} C_VEL
LIN {X 0,Y 214.238,Z 413.796,A -85,B 0,C 180,E1 -20797.533,E2 -20797.533} C_VEL
LIN {X 0,Y 214.036,Z 413.822,A -85,B 0,C 180,E1 -20801.355,E2 -20801.355} C_VEL
LIN {X 0,Y 213.92,Z 413.835,A -85,B 0,C 180,E1 -20805.23,E2 -20805.23} C_VEL
LIN {X 0,Y 213.821,Z 413.848,A -85,B 0,C 180,E1 -20809.181,E2 -20809.181} C_VEL
LIN {X 0,Y 213.741,Z 413.858,A -85,B 0,C 180,E1 -20813.231,E2 -20813.231} C_VEL
LIN {X 0,Y 213.531,Z 413.886,A -85,B 0,C 180,E1 -20817.429,E2 -20817.429} C_VEL
LIN {X 0,Y 212.976,Z 413.957,A -85,B 0,C 180,E1 -20821.86,E2 -20821.86} C_VEL
LIN {X 0,Y 212.769,Z 414.174,A -85,B 0,C 180,E1 -20824.009,E2 -20824.009} C_VEL
LIN {X 0,Y 215.56,Z 424.758,A -85,B 0,C 180,E1 -20825.065,E2 -20825.065} C_VEL
LIN {X 0,Y 218.231,Z 437.15,A -85,B 0,C 180,E1 -20826.557,E2 -20826.557} C_VEL
LIN {X 0,Y 220.285,Z 448.292,A -85,B 0,C 180,E1 -20828.171,E2 -20828.171} C_VEL
LIN {X 0,Y 220.799,Z 451.223,A -85,B 0,C 180,E1 -20828.647,E2 -20828.647} C_VEL
LIN {X 0,Y 220.172,Z 457.161,A -85,B 0,C 180,E1 -20829.581,E2 -20829.581} C_VEL
LIN {X 0,Y 218.4,Z 468.066,A -85,B 0,C 180,E1 -20831.571,E2 -20831.571} C_VEL
LIN {X 0,Y 216.805,Z 478.037,A -85,B 0,C 180,E1 -20833.844,E2 -20833.844} C_VEL
LIN {X 0,Y 215.041,Z 487.978,A -85,B 0,C 180,E1 -20836.663,E2 -20836.663} C_VEL
LIN {X 0,Y 213.724,Z 496.191,A -85,B 0,C 180,E1 -20839.594,E2 -20839.594} C_VEL
LIN {X 0,Y 212.768,Z 502.531,A -85,B 0,C 180,E1 -20842.43,E2 -20842.43} C_VEL
LIN {X 0,Y 212.067,Z 508.29,A -85,B 0,C 180,E1 -20845.712,E2 -20845.712} C_VEL
LIN {X 0,Y 211.617,Z 512.488,A -85,B 0,C 180,E1 -20848.904,E2 -20848.904} C_VEL
LIN {X 0,Y 211.479,Z 515.536,A -85,B 0,C 180,E1 -20852.275,E2 -20852.275} C_VEL
LIN {X 0,Y 211.683,Z 516.809,A -85,B 0,C 180,E1 -20854.432,E2 -20854.432} C_VEL
LIN {X 0,Y 212.344,Z 517.835,A -85,B 0,C 180,E1 -20857.906,E2 -20857.906} C_VEL
LIN {X 0,Y 213.337,Z 517.679,A -85,B 0,C 180,E1 -20860.768,E2 -20860.768} C_VEL
LIN {X 0,Y 214.315,Z 517.032,A -85,B 0,C 180,E1 -20862.836,E2 -20862.836} C_VEL
LIN {X 0,Y 216.667,Z 514.521,A -85,B 0,C 180,E1 -20866.644,E2 -20866.644} C_VEL
LIN {X 0,Y 219.319,Z 511.055,A -85,B 0,C 180,E1 -20869.851,E2 -20869.851} C_VEL
LIN {X 0,Y 222.341,Z 506.62,A -85,B 0,C 180,E1 -20872.738,E2 -20872.738} C_VEL
LIN {X 0,Y 226.42,Z 499.991,A -85,B 0,C 180,E1 -20875.89,E2 -20875.89} C_VEL
LIN {X 0,Y 230.598,Z 492.539,A -85,B 0,C 180,E1 -20878.613,E2 -20878.613} C_VEL
LIN {X 0,Y 234.625,Z 484.616,A -85,B 0,C 180,E1 -20880.86,E2 -20880.86} C_VEL
LIN {X 0,Y 238.69,Z 475.413,A -85,B 0,C 180,E1 -20882.955,E2 -20882.955} C_VEL
LIN {X 0,Y 238.188,Z 465.44,A -85,B 0,C 180,E1 -20886.184,E2 -20886.184} C_VEL
LIN {X 0,Y 237.45,Z 460.906,A -85,B 0,C 180,E1 -20887.717,E2 -20887.717} C_VEL
LIN {X 0,Y 235.536,Z 454.139,A -85,B 0,C 180,E1 -20890.315,E2 -20890.315} C_VEL
LIN {X 0,Y 233.347,Z 448.821,A -85,B 0,C 180,E1 -20892.758,E2 -20892.758} C_VEL
LIN {X 0,Y 230.338,Z 443.394,A -85,B 0,C 180,E1 -20895.94,E2 -20895.94} C_VEL
LIN {X 0,Y 228.615,Z 440.603,A -85,B 0,C 180,E1 -20897.905,E2 -20897.905} C_VEL
LIN {X 0,Y 224.575,Z 435.244,A -85,B 0,C 180,E1 -20904.007,E2 -20904.007} C_VEL
LIN {X 0,Y 222.954,Z 434.781,A -85,B 0,C 180,E1 -20908.22,E2 -20908.22} C_VEL
LIN {X 0,Y 222.725,Z 435.301,A -85,B 0,C 180,E1 -20911.589,E2 -20911.589} C_VEL
LIN {X 0,Y 223.408,Z 437.07,A -85,B 0,C 180,E1 -20915.138,E2 -20915.138} C_VEL
LIN {X 0,Y 225.28,Z 439.655,A -85,B 0,C 180,E1 -20918.76,E2 -20918.76} C_VEL
LIN {X 0,Y 225.927,Z 441.693,A -85,B 0,C 180,E1 -20920.138,E2 -20920.138} C_VEL
LIN {X 0,Y 227.804,Z 445.677,A -85,B 0,C 180,E1 -20922.746,E2 -20922.746} C_VEL
LIN {X 0,Y 228.544,Z 446.646,A -85,B 0,C 180,E1 -20923.498,E2 -20923.498} C_VEL
LIN {X 0,Y 231.335,Z 453.716,A -85,B 0,C 180,E1 -20926.815,E2 -20926.815} C_VEL
LIN {X 0,Y 233.119,Z 459.229,A -85,B 0,C 180,E1 -20928.913,E2 -20928.913} C_VEL
LIN {X 0,Y 233.992,Z 463.299,A -85,B 0,C 180,E1 -20930.231,E2 -20930.231} C_VEL
LIN {X 0,Y 234.727,Z 472.849,A -85,B 0,C 180,E1 -20932.812,E2 -20932.812} C_VEL
LIN {X 0,Y 234.83,Z 480.961,A -85,B 0,C 180,E1 -20934.912,E2 -20934.912} C_VEL
LIN {X 0,Y 234.192,Z 488.536,A -85,B 0,C 180,E1 -20936.833,E2 -20936.833} C_VEL
LIN {X 0,Y 232.942,Z 492.885,A -85,B 0,C 180,E1 -20937.793,E2 -20937.793} C_VEL
LIN {X 0,Y 230.67,Z 497.292,A -85,B 0,C 180,E1 -20938.624,E2 -20938.624} C_VEL
LIN {X 0,Y 224.889,Z 505.709,A -85,B 0,C 180,E1 -20940.245,E2 -20940.245} C_VEL
LIN {X 0,Y 222.299,Z 509.597,A -85,B 0,C 180,E1 -20941.217,E2 -20941.217} C_VEL
LIN {X 0,Y 221.61,Z 510.805,A -85,B 0,C 180,E1 -20941.584,E2 -20941.584} C_VEL
LIN {X 0,Y 216.792,Z 519.293,A -85,B 0,C 180,E1 -20944.57,E2 -20944.57} C_VEL
LIN {X 0,Y 212.938,Z 525.763,A -85,B 0,C 180,E1 -20947.542,E2 -20947.542} C_VEL
LIN {X 0,Y 210.194,Z 530.638,A -85,B 0,C 180,E1 -20950.475,E2 -20950.475} C_VEL
LIN {X 0,Y 207.289,Z 535.245,A -85,B 0,C 180,E1 -20954.27,E2 -20954.27} C_VEL
LIN {X 0,Y 205.469,Z 538.319,A -85,B 0,C 180,E1 -20958.165,E2 -20958.165} C_VEL
LIN {X 0,Y 204.644,Z 539.832,A -85,B 0,C 180,E1 -20962.112,E2 -20962.112} C_VEL
LIN {X 0,Y 204.599,Z 539.858,A -85,B 0,C 180,E1 -20966.068,E2 -20966.068} C_VEL
LIN {X 0,Y 204.702,Z 539.296,A -85,B 0,C 180,E1 -20968.04,E2 -20968.04} C_VEL
LIN {X 0,Y 204.841,Z 538.283,A -85,B 0,C 180,E1 -20970.007,E2 -20970.007} C_VEL
LIN {X 0,Y 204.776,Z 536.818,A -85,B 0,C 180,E1 -20971.974,E2 -20971.974} C_VEL
LIN {X 0,Y 204.861,Z 533.776,A -85,B 0,C 180,E1 -20974.935,E2 -20974.935} C_VEL
LIN {X 0,Y 204.946,Z 529.617,A -85,B 0,C 180,E1 -20977.891,E2 -20977.891} C_VEL
LIN {X 0,Y 205.46,Z 523.229,A -85,B 0,C 180,E1 -20981.35,E2 -20981.35} C_VEL
LIN {X 0,Y 206.417,Z 516.196,A -85,B 0,C 180,E1 -20984.298,E2 -20984.298} C_VEL
LIN {X 0,Y 207.737,Z 507.436,A -85,B 0,C 180,E1 -20987.226,E2 -20987.226} C_VEL
LIN {X 0,Y 209.459,Z 497.747,A -85,B 0,C 180,E1 -20989.819,E2 -20989.819} C_VEL
LIN {X 0,Y 211.008,Z 488.83,A -85,B 0,C 180,E1 -20991.756,E2 -20991.756} C_VEL
LIN {X 0,Y 210.522,Z 477.594,A -85,B 0,C 180,E1 -20993.836,E2 -20993.836} C_VEL
LIN {X 0,Y 209.622,Z 465.267,A -85,B 0,C 180,E1 -20995.718,E2 -20995.718} C_VEL
LIN {X 0,Y 208.413,Z 451.776,A -85,B 0,C 180,E1 -20997.338,E2 -20997.338} C_VEL
LIN {X 0,Y 206.898,Z 438.363,A -85,B 0,C 180,E1 -20998.584,E2 -20998.584} C_VEL
LIN {X 0,Y 206.604,Z 435.42,A -85,B 0,C 180,E1 -20998.794,E2 -20998.794} C_VEL
LIN {X 0,Y 207.965,Z 430.036,A -85,B 0,C 180,E1 -21003.897,E2 -21003.897} C_VEL
LIN {X 0,Y 208.602,Z 427.789,A -85,B 0,C 180,E1 -21006.04,E2 -21006.04} C_VEL
LIN {X 0,Y 208.775,Z 426.499,A -85,B 0,C 180,E1 -21007.304,E2 -21007.304} C_VEL
LIN {X 0,Y 208.592,Z 423.998,A -85,B 0,C 180,E1 -21009.811,E2 -21009.811} C_VEL
LIN {X 0,Y 207.639,Z 419.364,A -85,B 0,C 180,E1 -21014.699,E2 -21014.699} C_VEL
LIN {X 0,Y 206.783,Z 414.725,A -85,B 0,C 180,E1 -21020.01,E2 -21020.01} C_VEL
LIN {X 0,Y 206.719,Z 414.732,A -85,B 0,C 180,E1 -21024.691,E2 -21024.691} C_VEL
LIN {X 0,Y 206.716,Z 414.736,A -85,B 0,C 180,E1 -21029.336,E2 -21029.336} C_VEL
LIN {X 0,Y 206.723,Z 414.73,A -85,B 0,C 180,E1 -21033.769,E2 -21033.769} C_VEL
LIN {X 0,Y 206.737,Z 414.731,A -85,B 0,C 180,E1 -21038.039,E2 -21038.039} C_VEL
LIN {X 0,Y 206.842,Z 414.715,A -85,B 0,C 180,E1 -21042.192,E2 -21042.192} C_VEL
LIN {X 0,Y 206.892,Z 414.712,A -85,B 0,C 180,E1 -21046.242,E2 -21046.242} C_VEL
LIN {X 0,Y 207.099,Z 414.682,A -85,B 0,C 180,E1 -21050.229,E2 -21050.229} C_VEL
LIN {X 0,Y 207.068,Z 414.69,A -85,B 0,C 180,E1 -21054.154,E2 -21054.154} C_VEL
LIN {X 0,Y 207.395,Z 414.646,A -85,B 0,C 180,E1 -21058.056,E2 -21058.056} C_VEL
LIN {X 0,Y 207.519,Z 414.632,A -85,B 0,C 180,E1 -21059.998,E2 -21059.998} C_VEL
LIN {X 0,Y 207.065,Z 414.69,A -85,B 0,C 180,E1 -21063.891,E2 -21063.891} C_VEL
LIN {X 0,Y 207.139,Z 414.679,A -85,B 0,C 180,E1 -21067.798,E2 -21067.798} C_VEL
LIN {X 0,Y 206.931,Z 414.707,A -85,B 0,C 180,E1 -21071.756,E2 -21071.756} C_VEL
LIN {X 0,Y 206.84,Z 414.715,A -85,B 0,C 180,E1 -21075.771,E2 -21075.771} C_VEL
LIN {X 0,Y 206.731,Z 414.732,A -85,B 0,C 180,E1 -21079.872,E2 -21079.872} C_VEL
LIN {X 0,Y 206.755,Z 414.726,A -85,B 0,C 180,E1 -21084.071,E2 -21084.071} C_VEL
LIN {X 0,Y 206.742,Z 414.733,A -85,B 0,C 180,E1 -21088.417,E2 -21088.417} C_VEL
LIN {X 0,Y 206.708,Z 414.735,A -85,B 0,C 180,E1 -21092.954,E2 -21092.954} C_VEL
LIN {X 0,Y 206.691,Z 414.736,A -85,B 0,C 180,E1 -21097.735,E2 -21097.735} C_VEL
LIN {X 0,Y 206.651,Z 414.74,A -85,B 0,C 180,E1 -21101.557,E2 -21101.557} C_VEL
LIN {X 0,Y 206.64,Z 414.743,A -85,B 0,C 180,E1 -21105.577,E2 -21105.577} C_VEL
LIN {X 0,Y 206.66,Z 414.739,A -85,B 0,C 180,E1 -21109.741,E2 -21109.741} C_VEL
LIN {X 0,Y 206.706,Z 414.736,A -85,B 0,C 180,E1 -21114.683,E2 -21114.683} C_VEL
LIN {X 0,Y 206.719,Z 414.733,A -85,B 0,C 180,E1 -21119.331,E2 -21119.331} C_VEL
LIN {X 0,Y 206.737,Z 414.73,A -85,B 0,C 180,E1 -21123.766,E2 -21123.766} C_VEL
LIN {X 0,Y 206.761,Z 414.729,A -85,B 0,C 180,E1 -21128.037,E2 -21128.037} C_VEL
LIN {X 0,Y 206.875,Z 414.715,A -85,B 0,C 180,E1 -21132.19,E2 -21132.19} C_VEL
LIN {X 0,Y 206.895,Z 414.714,A -85,B 0,C 180,E1 -21136.237,E2 -21136.237} C_VEL
LIN {X 0,Y 207.097,Z 414.688,A -85,B 0,C 180,E1 -21140.224,E2 -21140.224} C_VEL
LIN {X 0,Y 207.057,Z 414.693,A -85,B 0,C 180,E1 -21144.149,E2 -21144.149} C_VEL
LIN {X 0,Y 207.376,Z 414.654,A -85,B 0,C 180,E1 -21148.051,E2 -21148.051} C_VEL
LIN {X 0,Y 207.508,Z 414.635,A -85,B 0,C 180,E1 -21149.993,E2 -21149.993} C_VEL
LIN {X 0,Y 207.376,Z 414.651,A -85,B 0,C 180,E1 -21151.935,E2 -21151.935} C_VEL
LIN {X 0,Y 207.179,Z 414.676,A -85,B 0,C 180,E1 -21157.791,E2 -21157.791} C_VEL
LIN {X 0,Y 206.972,Z 414.703,A -85,B 0,C 180,E1 -21161.748,E2 -21161.748} C_VEL
LIN {X 0,Y 206.854,Z 414.717,A -85,B 0,C 180,E1 -21165.764,E2 -21165.764} C_VEL
LIN {X 0,Y 206.762,Z 414.73,A -85,B 0,C 180,E1 -21169.863,E2 -21169.863} C_VEL
LIN {X 0,Y 206.627,Z 414.747,A -85,B 0,C 180,E1 -21174.08,E2 -21174.08} C_VEL
LIN {X 0,Y 206.318,Z 414.785,A -85,B 0,C 180,E1 -21178.474,E2 -21178.474} C_VEL
LIN {X 0,Y 205.8,Z 414.852,A -85,B 0,C 180,E1 -21183.11,E2 -21183.11} C_VEL
LIN {X 0,Y 205.769,Z 414.855,A -85,B 0,C 180,E1 -21183.408,E2 -21183.408} C_VEL
LIN {X 0,Y 208.675,Z 425.99,A -85,B 0,C 180,E1 -21184.624,E2 -21184.624} C_VEL
LIN {X 0,Y 211.639,Z 439.852,A -85,B 0,C 180,E1 -21186.402,E2 -21186.402} C_VEL
LIN {X 0,Y 213.826,Z 452.27,A -85,B 0,C 180,E1 -21188.357,E2 -21188.357} C_VEL
LIN {X 0,Y 212.654,Z 460.875,A -85,B 0,C 180,E1 -21189.794,E2 -21189.794} C_VEL
LIN {X 0,Y 210.703,Z 472.74,A -85,B 0,C 180,E1 -21192.222,E2 -21192.222} C_VEL
LIN {X 0,Y 209.122,Z 481.705,A -85,B 0,C 180,E1 -21194.498,E2 -21194.498} C_VEL
LIN {X 0,Y 207.537,Z 490.833,A -85,B 0,C 180,E1 -21197.371,E2 -21197.371} C_VEL
LIN {X 0,Y 206.364,Z 498.246,A -85,B 0,C 180,E1 -21200.264,E2 -21200.264} C_VEL
LIN {X 0,Y 205.463,Z 504.358,A -85,B 0,C 180,E1 -21203.233,E2 -21203.233} C_VEL
LIN {X 0,Y 204.824,Z 509.863,A -85,B 0,C 180,E1 -21206.704,E2 -21206.704} C_VEL
LIN {X 0,Y 204.488,Z 512.924,A -85,B 0,C 180,E1 -21209.212,E2 -21209.212} C_VEL
LIN {X 0,Y 204.362,Z 514.827,A -85,B 0,C 180,E1 -21211.221,E2 -21211.221} C_VEL
LIN {X 0,Y 204.494,Z 516.46,A -85,B 0,C 180,E1 -21213.465,E2 -21213.465} C_VEL
LIN {X 0,Y 204.76,Z 517.591,A -85,B 0,C 180,E1 -21215.679,E2 -21215.679} C_VEL
LIN {X 0,Y 205.241,Z 518.186,A -85,B 0,C 180,E1 -21217.875,E2 -21217.875} C_VEL
LIN {X 0,Y 205.937,Z 518.334,A -85,B 0,C 180,E1 -21220.048,E2 -21220.048} C_VEL
LIN {X 0,Y 206.846,Z 517.998,A -85,B 0,C 180,E1 -21222.196,E2 -21222.196} C_VEL
LIN {X 0,Y 207.994,Z 517.189,A -85,B 0,C 180,E1 -21224.319,E2 -21224.319} C_VEL
LIN {X 0,Y 209.488,Z 515.829,A -85,B 0,C 180,E1 -21226.594,E2 -21226.594} C_VEL
LIN {X 0,Y 211.816,Z 513.198,A -85,B 0,C 180,E1 -21229.487,E2 -21229.487} C_VEL
LIN {X 0,Y 214.788,Z 509.321,A -85,B 0,C 180,E1 -21232.481,E2 -21232.481} C_VEL
LIN {X 0,Y 218.512,Z 504.004,A -85,B 0,C 180,E1 -21235.489,E2 -21235.489} C_VEL
LIN {X 0,Y 223.246,Z 496.545,A -85,B 0,C 180,E1 -21238.631,E2 -21238.631} C_VEL
LIN {X 0,Y 227.114,Z 489.64,A -85,B 0,C 180,E1 -21240.888,E2 -21240.888} C_VEL
LIN {X 0,Y 232.264,Z 479.493,A -85,B 0,C 180,E1 -21243.471,E2 -21243.471} C_VEL
LIN {X 0,Y 232.997,Z 477.867,A -85,B 0,C 180,E1 -21243.849,E2 -21243.849} C_VEL
LIN {X 0,Y 232.832,Z 468.954,A -85,B 0,C 180,E1 -21246.936,E2 -21246.936} C_VEL
LIN {X 0,Y 232.214,Z 464.243,A -85,B 0,C 180,E1 -21248.705,E2 -21248.705} C_VEL
LIN {X 0,Y 230.65,Z 458.181,A -85,B 0,C 180,E1 -21251.281,E2 -21251.281} C_VEL
LIN {X 0,Y 228.847,Z 453.629,A -85,B 0,C 180,E1 -21253.612,E2 -21253.612} C_VEL
LIN {X 0,Y 226.841,Z 449.477,A -85,B 0,C 180,E1 -21256.199,E2 -21256.199} C_VEL
LIN {X 0,Y 225.363,Z 446.885,A -85,B 0,C 180,E1 -21258.172,E2 -21258.172} C_VEL
LIN {X 0,Y 222.176,Z 442.319,A -85,B 0,C 180,E1 -21263.48,E2 -21263.48} C_VEL
LIN {X 0,Y 221.876,Z 441.805,A -85,B 0,C 180,E1 -21264.318,E2 -21264.318} C_VEL
LIN {X 0,Y 220.467,Z 441.483,A -85,B 0,C 180,E1 -21268.567,E2 -21268.567} C_VEL
LIN {X 0,Y 220.269,Z 441.74,A -85,B 0,C 180,E1 -21270.699,E2 -21270.699} C_VEL
LIN {X 0,Y 220.648,Z 443.126,A -85,B 0,C 180,E1 -21274.106,E2 -21274.106} C_VEL
LIN {X 0,Y 222.04,Z 445.534,A -85,B 0,C 180,E1 -21277.706,E2 -21277.706} C_VEL
LIN {X 0,Y 222.767,Z 446.965,A -85,B 0,C 180,E1 -21279.124,E2 -21279.124} C_VEL
LIN {X 0,Y 224.529,Z 451.718,A -85,B 0,C 180,E1 -21282.299,E2 -21282.299} C_VEL
LIN {X 0,Y 225.287,Z 453.24,A -85,B 0,C 180,E1 -21283.34,E2 -21283.34} C_VEL
LIN {X 0,Y 227.488,Z 459.879,A -85,B 0,C 180,E1 -21286.541,E2 -21286.541} C_VEL
LIN {X 0,Y 228.788,Z 464.435,A -85,B 0,C 180,E1 -21288.382,E2 -21288.382} C_VEL
LIN {X 0,Y 229.373,Z 469.397,A -85,B 0,C 180,E1 -21289.998,E2 -21289.998} C_VEL
LIN {X 0,Y 229.5,Z 480.061,A -85,B 0,C 180,E1 -21293.034,E2 -21293.034} C_VEL
LIN {X 0,Y 228.763,Z 488.656,A -85,B 0,C 180,E1 -21295.375,E2 -21295.375} C_VEL
LIN {X 0,Y 226.981,Z 497.889,A -85,B 0,C 180,E1 -21297.913,E2 -21297.913} C_VEL
LIN {X 0,Y 224.59,Z 505.128,A -85,B 0,C 180,E1 -21299.964,E2 -21299.964} C_VEL
LIN {X 0,Y 221.61,Z 510.805,A -85,B 0,C 180,E1 -21301.584,E2 -21301.584} C_VEL
LIN {X 0,Y 219.139,Z 514.378,A -85,B 0,C 180,E1 -21302.639,E2 -21302.639} C_VEL
LIN {X 0,Y 213.476,Z 519.876,A -85,B 0,C 180,E1 -21304.251,E2 -21304.251} C_VEL
LIN {X 0,Y 207.961,Z 524.672,A -85,B 0,C 180,E1 -21306.052,E2 -21306.052} C_VEL
LIN {X 0,Y 205.773,Z 527.193,A -85,B 0,C 180,E1 -21307.382,E2 -21307.382} C_VEL
LIN {X 0,Y 202.7,Z 532.106,A -85,B 0,C 180,E1 -21310.777,E2 -21310.777} C_VEL
LIN {X 0,Y 200.432,Z 535.261,A -85,B 0,C 180,E1 -21313.717,E2 -21313.717} C_VEL
LIN {X 0,Y 199.277,Z 536.873,A -85,B 0,C 180,E1 -21315.716,E2 -21315.716} C_VEL
LIN {X 0,Y 197.938,Z 538.946,A -85,B 0,C 180,E1 -21319.782,E2 -21319.782} C_VEL
LIN {X 0,Y 197.486,Z 539.568,A -85,B 0,C 180,E1 -21323.879,E2 -21323.879} C_VEL
LIN {X 0,Y 197.525,Z 539.303,A -85,B 0,C 180,E1 -21325.927,E2 -21325.927} C_VEL
LIN {X 0,Y 197.632,Z 538.618,A -85,B 0,C 180,E1 -21327.97,E2 -21327.97} C_VEL
LIN {X 0,Y 197.773,Z 537.534,A -85,B 0,C 180,E1 -21330.007,E2 -21330.007} C_VEL
LIN {X 0,Y 197.712,Z 536.008,A -85,B 0,C 180,E1 -21332.045,E2 -21332.045} C_VEL
LIN {X 0,Y 197.79,Z 534.042,A -85,B 0,C 180,E1 -21334.083,E2 -21334.083} C_VEL
LIN {X 0,Y 197.817,Z 530.11,A -85,B 0,C 180,E1 -21337.15,E2 -21337.15} C_VEL
LIN {X 0,Y 198.144,Z 524.962,A -85,B 0,C 180,E1 -21340.222,E2 -21340.222} C_VEL
LIN {X 0,Y 198.89,Z 518.459,A -85,B 0,C 180,E1 -21343.286,E2 -21343.286} C_VEL
LIN {X 0,Y 200.206,Z 510.41,A -85,B 0,C 180,E1 -21346.317,E2 -21346.317} C_VEL
LIN {X 0,Y 201.47,Z 502.166,A -85,B 0,C 180,E1 -21348.832,E2 -21348.832} C_VEL
LIN {X 0,Y 203.367,Z 492.207,A -85,B 0,C 180,E1 -21351.282,E2 -21351.282} C_VEL
LIN {X 0,Y 203.969,Z 488.807,A -85,B 0,C 180,E1 -21352.013,E2 -21352.013} C_VEL
LIN {X 0,Y 203.463,Z 477.343,A -85,B 0,C 180,E1 -21354.224,E2 -21354.224} C_VEL
LIN {X 0,Y 202.63,Z 465.539,A -85,B 0,C 180,E1 -21356.104,E2 -21356.104} C_VEL
LIN {X 0,Y 201.554,Z 452.92,A -85,B 0,C 180,E1 -21357.718,E2 -21357.718} C_VEL
LIN {X 0,Y 200.022,Z 438.658,A -85,B 0,C 180,E1 -21359.124,E2 -21359.124} C_VEL
LIN {X 0,Y 199.668,Z 435.02,A -85,B 0,C 180,E1 -21359.434,E2 -21359.434} C_VEL
LIN {X 0,Y 201.229,Z 429.174,A -85,B 0,C 180,E1 -21365.196,E2 -21365.196} C_VEL
LIN {X 0,Y 201.667,Z 426.697,A -85,B 0,C 180,E1 -21367.681,E2 -21367.681} C_VEL
LIN {X 0,Y 201.506,Z 424.59,A -85,B 0,C 180,E1 -21369.885,E2 -21369.885} C_VEL
LIN {X 0,Y 200.641,Z 420.376,A -85,B 0,C 180,E1 -21374.48,E2 -21374.48} C_VEL
LIN {X 0,Y 199.741,Z 415.603,A -85,B 0,C 180,E1 -21380.006,E2 -21380.006} C_VEL
LIN {X 0,Y 199.634,Z 415.613,A -85,B 0,C 180,E1 -21384.077,E2 -21384.077} C_VEL
LIN {X 0,Y 199.705,Z 415.607,A -85,B 0,C 180,E1 -21388.136,E2 -21388.136} C_VEL
LIN {X 0,Y 199.662,Z 415.612,A -85,B 0,C 180,E1 -21392.766,E2 -21392.766} C_VEL
LIN {X 0,Y 199.698,Z 415.611,A -85,B 0,C 180,E1 -21397.223,E2 -21397.223} C_VEL
LIN {X 0,Y 199.766,Z 415.596,A -85,B 0,C 180,E1 -21401.803,E2 -21401.803} C_VEL
LIN {X 0,Y 199.829,Z 415.592,A -85,B 0,C 180,E1 -21405.746,E2 -21405.746} C_VEL
LIN {X 0,Y 200.044,Z 415.561,A -85,B 0,C 180,E1 -21409.881,E2 -21409.881} C_VEL
LIN {X 0,Y 200.031,Z 415.567,A -85,B 0,C 180,E1 -21413.948,E2 -21413.948} C_VEL
LIN {X 0,Y 200.334,Z 415.525,A -85,B 0,C 180,E1 -21417.988,E2 -21417.988} C_VEL
LIN {X 0,Y 200.484,Z 415.508,A -85,B 0,C 180,E1 -21419.998,E2 -21419.998} C_VEL
LIN {X 0,Y 200.011,Z 415.569,A -85,B 0,C 180,E1 -21424.028,E2 -21424.028} C_VEL
LIN {X 0,Y 200.087,Z 415.557,A -85,B 0,C 180,E1 -21428.075,E2 -21428.075} C_VEL
LIN {X 0,Y 199.881,Z 415.586,A -85,B 0,C 180,E1 -21432.177,E2 -21432.177} C_VEL
LIN {X 0,Y 199.778,Z 415.596,A -85,B 0,C 180,E1 -21436.344,E2 -21436.344} C_VEL
LIN {X 0,Y 199.663,Z 415.615,A -85,B 0,C 180,E1 -21440.607,E2 -21440.607} C_VEL
LIN {X 0,Y 199.676,Z 415.612,A -85,B 0,C 180,E1 -21444.982,E2 -21444.982} C_VEL
LIN {X 0,Y 199.671,Z 415.611,A -85,B 0,C 180,E1 -21449.521,E2 -21449.521} C_VEL
LIN {X 0,Y 199.679,Z 415.608,A -85,B 0,C 180,E1 -21452.348,E2 -21452.348} C_VEL
LIN {X 0,Y 199.635,Z 415.618,A -85,B 0,C 180,E1 -21456.758,E2 -21456.758} C_VEL
LIN {X 0,Y 199.619,Z 415.615,A -85,B 0,C 180,E1 -21459.323,E2 -21459.323} C_VEL
LIN {X 0,Y 199.583,Z 415.622,A -85,B 0,C 180,E1 -21462.304,E2 -21462.304} C_VEL
LIN {X 0,Y 199.587,Z 415.622,A -85,B 0,C 180,E1 -21465.222,E2 -21465.222} C_VEL
LIN {X 0,Y 199.583,Z 415.621,A -85,B 0,C 180,E1 -21467.998,E2 -21467.998} C_VEL
LIN {X 0,Y 199.609,Z 415.621,A -85,B 0,C 180,E1 -21470.765,E2 -21470.765} C_VEL
LIN {X 0,Y 199.619,Z 415.616,A -85,B 0,C 180,E1 -21475.707,E2 -21475.707} C_VEL
LIN {X 0,Y 199.699,Z 415.606,A -85,B 0,C 180,E1 -21478.129,E2 -21478.129} C_VEL
LIN {X 0,Y 199.692,Z 415.609,A -85,B 0,C 180,E1 -21482.765,E2 -21482.765} C_VEL
LIN {X 0,Y 199.741,Z 415.602,A -85,B 0,C 180,E1 -21487.222,E2 -21487.222} C_VEL
LIN {X 0,Y 199.798,Z 415.595,A -85,B 0,C 180,E1 -21491.75,E2 -21491.75} C_VEL
LIN {X 0,Y 199.836,Z 415.59,A -85,B 0,C 180,E1 -21495.741,E2 -21495.741} C_VEL
LIN {X 0,Y 200.02,Z 415.569,A -85,B 0,C 180,E1 -21499.874,E2 -21499.874} C_VEL
LIN {X 0,Y 200.019,Z 415.568,A -85,B 0,C 180,E1 -21503.942,E2 -21503.942} C_VEL
LIN {X 0,Y 200.315,Z 415.533,A -85,B 0,C 180,E1 -21507.982,E2 -21507.982} C_VEL
LIN {X 0,Y 200.473,Z 415.511,A -85,B 0,C 180,E1 -21509.993,E2 -21509.993} C_VEL
LIN {X 0,Y 200.025,Z 415.57,A -85,B 0,C 180,E1 -21514.022,E2 -21514.022} C_VEL
LIN {X 0,Y 200.122,Z 415.555,A -85,B 0,C 180,E1 -21518.068,E2 -21518.068} C_VEL
LIN {X 0,Y 199.903,Z 415.586,A -85,B 0,C 180,E1 -21522.17,E2 -21522.17} C_VEL
LIN {X 0,Y 199.791,Z 415.594,A -85,B 0,C 180,E1 -21526.336,E2 -21526.336} C_VEL
LIN {X 0,Y 199.665,Z 415.613,A -85,B 0,C 180,E1 -21530.6,E2 -21530.6} C_VEL
LIN {X 0,Y 199.526,Z 415.629,A -85,B 0,C 180,E1 -21534.995,E2 -21534.995} C_VEL
LIN {X 0,Y 199.307,Z 415.66,A -85,B 0,C 180,E1 -21538.174,E2 -21538.174} C_VEL
LIN {X 0,Y 198.78,Z 415.726,A -85,B 0,C 180,E1 -21542.843,E2 -21542.843} C_VEL
LIN {X 0,Y 201.817,Z 427.181,A -85,B 0,C 180,E1 -21544.152,E2 -21544.152} C_VEL
LIN {X 0,Y 204.695,Z 440.795,A -85,B 0,C 180,E1 -21545.986,E2 -21545.986} C_VEL
LIN {X 0,Y 206.856,Z 453.172,A -85,B 0,C 180,E1 -21548.03,E2 -21548.03} C_VEL
LIN {X 0,Y 205.363,Z 463.207,A -85,B 0,C 180,E1 -21549.803,E2 -21549.803} C_VEL
LIN {X 0,Y 203.58,Z 473.75,A -85,B 0,C 180,E1 -21552.082,E2 -21552.082} C_VEL
LIN {X 0,Y 201.911,Z 482.88,A -85,B 0,C 180,E1 -21554.523,E2 -21554.523} C_VEL
LIN {X 0,Y 200.36,Z 491.703,A -85,B 0,C 180,E1 -21557.431,E2 -21557.431} C_VEL
LIN {X 0,Y 199.145,Z 499.323,A -85,B 0,C 180,E1 -21560.565,E2 -21560.565} C_VEL
LIN {X 0,Y 198.208,Z 505.714,A -85,B 0,C 180,E1 -21563.913,E2 -21563.913} C_VEL
LIN {X 0,Y 197.587,Z 511.3,A -85,B 0,C 180,E1 -21567.758,E2 -21567.758} C_VEL
LIN {X 0,Y 197.273,Z 514.955,A -85,B 0,C 180,E1 -21571.255,E2 -21571.255} C_VEL
LIN {X 0,Y 197.51,Z 517.344,A -85,B 0,C 180,E1 -21574.725,E2 -21574.725} C_VEL
LIN {X 0,Y 197.998,Z 518.381,A -85,B 0,C 180,E1 -21577.327,E2 -21577.327} C_VEL
LIN {X 0,Y 198.54,Z 518.767,A -85,B 0,C 180,E1 -21579.271,E2 -21579.271} C_VEL
LIN {X 0,Y 199.589,Z 518.691,A -85,B 0,C 180,E1 -21581.911,E2 -21581.911} C_VEL
LIN {X 0,Y 201.846,Z 517.365,A -85,B 0,C 180,E1 -21585.895,E2 -21585.895} C_VEL
LIN {X 0,Y 203.368,Z 515.967,A -85,B 0,C 180,E1 -21588.035,E2 -21588.035} C_VEL
LIN {X 0,Y 206.195,Z 512.964,A -85,B 0,C 180,E1 -21591.222,E2 -21591.222} C_VEL
LIN {X 0,Y 209.557,Z 508.922,A -85,B 0,C 180,E1 -21594.227,E2 -21594.227} C_VEL
LIN {X 0,Y 213.513,Z 503.578,A -85,B 0,C 180,E1 -21597.172,E2 -21597.172} C_VEL
LIN {X 0,Y 218.012,Z 496.857,A -85,B 0,C 180,E1 -21600.002,E2 -21600.002} C_VEL
LIN {X 0,Y 223.058,Z 488.423,A -85,B 0,C 180,E1 -21602.71,E2 -21602.71} C_VEL
LIN {X 0,Y 227.291,Z 480.291,A -85,B 0,C 180,E1 -21604.794,E2 -21604.794} C_VEL
LIN {X 0,Y 227.511,Z 471.771,A -85,B 0,C 180,E1 -21607.993,E2 -21607.993} C_VEL
LIN {X 0,Y 226.534,Z 465.424,A -85,B 0,C 180,E1 -21610.729,E2 -21610.729} C_VEL
LIN {X 0,Y 225.143,Z 460.27,A -85,B 0,C 180,E1 -21613.298,E2 -21613.298} C_VEL
LIN {X 0,Y 223.065,Z 455.395,A -85,B 0,C 180,E1 -21616.474,E2 -21616.474} C_VEL
LIN {X 0,Y 221.849,Z 452.937,A -85,B 0,C 180,E1 -21618.471,E2 -21618.471} C_VEL
LIN {X 0,Y 219.617,Z 449.459,A -85,B 0,C 180,E1 -21622.584,E2 -21622.584} C_VEL
LIN {X 0,Y 218.847,Z 448.254,A -85,B 0,C 180,E1 -21624.677,E2 -21624.677} C_VEL
LIN {X 0,Y 217.614,Z 448.099,A -85,B 0,C 180,E1 -21629.327,E2 -21629.327} C_VEL
LIN {X 0,Y 217.711,Z 449.292,A -85,B 0,C 180,E1 -21633.285,E2 -21633.285} C_VEL
LIN {X 0,Y 219.058,Z 451.963,A -85,B 0,C 180,E1 -21637.561,E2 -21637.561} C_VEL
LIN {X 0,Y 219.647,Z 453.758,A -85,B 0,C 180,E1 -21639.098,E2 -21639.098} C_VEL
LIN {X 0,Y 221.744,Z 459.706,A -85,B 0,C 180,E1 -21643.212,E2 -21643.212} C_VEL
LIN {X 0,Y 223.433,Z 465.671,A -85,B 0,C 180,E1 -21646.222,E2 -21646.222} C_VEL
LIN {X 0,Y 224.252,Z 469.548,A -85,B 0,C 180,E1 -21647.863,E2 -21647.863} C_VEL
LIN {X 0,Y 224.488,Z 474.351,A -85,B 0,C 180,E1 -21649.472,E2 -21649.472} C_VEL
LIN {X 0,Y 223.993,Z 484.649,A -85,B 0,C 180,E1 -21652.603,E2 -21652.603} C_VEL
LIN {X 0,Y 222.5,Z 494.041,A -85,B 0,C 180,E1 -21655.36,E2 -21655.36} C_VEL
LIN {X 0,Y 220.337,Z 502.021,A -85,B 0,C 180,E1 -21657.715,E2 -21657.715} C_VEL
LIN {X 0,Y 218.56,Z 506.409,A -85,B 0,C 180,E1 -21659.045,E2 -21659.045} C_VEL
LIN {X 0,Y 213.242,Z 515.569,A -85,B 0,C 180,E1 -21661.997,E2 -21661.997} C_VEL
LIN {X 0,Y 208.527,Z 522.956,A -85,B 0,C 180,E1 -21665.093,E2 -21665.093} C_VEL
LIN {X 0,Y 205.773,Z 527.193,A -85,B 0,C 180,E1 -21667.382,E2 -21667.382} C_VEL
LIN {X 0,Y 203.709,Z 529.544,A -85,B 0,C 180,E1 -21668.79,E2 -21668.79} C_VEL
LIN {X 0,Y 198.763,Z 532.878,A -85,B 0,C 180,E1 -21671.054,E2 -21671.054} C_VEL
LIN {X 0,Y 194.053,Z 535.484,A -85,B 0,C 180,E1 -21673.486,E2 -21673.486} C_VEL
LIN {X 0,Y 192.406,Z 536.675,A -85,B 0,C 180,E1 -21675.122,E2 -21675.122} C_VEL
LIN {X 0,Y 190.935,Z 538.638,A -85,B 0,C 180,E1 -21679.403,E2 -21679.403} C_VEL
LIN {X 0,Y 190.563,Z 539.046,A -85,B 0,C 180,E1 -21681.525,E2 -21681.525} C_VEL
LIN {X 0,Y 190.456,Z 538.692,A -85,B 0,C 180,E1 -21685.776,E2 -21685.776} C_VEL
LIN {X 0,Y 190.564,Z 537.934,A -85,B 0,C 180,E1 -21687.894,E2 -21687.894} C_VEL
LIN {X 0,Y 190.706,Z 536.776,A -85,B 0,C 180,E1 -21690.008,E2 -21690.008} C_VEL
LIN {X 0,Y 190.67,Z 534.15,A -85,B 0,C 180,E1 -21693.177,E2 -21693.177} C_VEL
LIN {X 0,Y 190.728,Z 530.449,A -85,B 0,C 180,E1 -21696.354,E2 -21696.354} C_VEL
LIN {X 0,Y 190.985,Z 525.572,A -85,B 0,C 180,E1 -21699.539,E2 -21699.539} C_VEL
LIN {X 0,Y 191.613,Z 519.391,A -85,B 0,C 180,E1 -21702.721,E2 -21702.721} C_VEL
LIN {X 0,Y 192.881,Z 511.677,A -85,B 0,C 180,E1 -21705.867,E2 -21705.867} C_VEL
LIN {X 0,Y 194.382,Z 502.023,A -85,B 0,C 180,E1 -21708.997,E2 -21708.997} C_VEL
LIN {X 0,Y 196.205,Z 492.932,A -85,B 0,C 180,E1 -21711.356,E2 -21711.356} C_VEL
LIN {X 0,Y 196.913,Z 488.764,A -85,B 0,C 180,E1 -21712.292,E2 -21712.292} C_VEL
LIN {X 0,Y 196.426,Z 477.389,A -85,B 0,C 180,E1 -21714.586,E2 -21714.586} C_VEL
LIN {X 0,Y 195.551,Z 464.602,A -85,B 0,C 180,E1 -21716.703,E2 -21716.703} C_VEL
LIN {X 0,Y 194.422,Z 451.294,A -85,B 0,C 180,E1 -21718.428,E2 -21718.428} C_VEL
LIN {X 0,Y 192.934,Z 437.07,A -85,B 0,C 180,E1 -21719.84,E2 -21719.84} C_VEL
LIN {X 0,Y 192.712,Z 434.644,A -85,B 0,C 180,E1 -21720.067,E2 -21720.067} C_VEL
LIN {X 0,Y 194.187,Z 429.462,A -85,B 0,C 180,E1 -21725.393,E2 -21725.393} C_VEL
LIN {X 0,Y 194.593,Z 427.084,A -85,B 0,C 180,E1 -21727.886,E2 -21727.886} C_VEL
LIN {X 0,Y 194.301,Z 424.549,A -85,B 0,C 180,E1 -21730.631,E2 -21730.631} C_VEL
LIN {X 0,Y 193.258,Z 419.623,A -85,B 0,C 180,E1 -21736.292,E2 -21736.292} C_VEL
LIN {X 0,Y 192.704,Z 416.479,A -85,B 0,C 180,E1 -21740.173,E2 -21740.173} C_VEL
LIN {X 0,Y 192.58,Z 416.492,A -85,B 0,C 180,E1 -21744.272,E2 -21744.272} C_VEL
LIN {X 0,Y 192.625,Z 416.49,A -85,B 0,C 180,E1 -21747.063,E2 -21747.063} C_VEL
LIN {X 0,Y 192.64,Z 416.486,A -85,B 0,C 180,E1 -21751.686,E2 -21751.686} C_VEL
LIN {X 0,Y 192.691,Z 416.481,A -85,B 0,C 180,E1 -21756.345,E2 -21756.345} C_VEL
LIN {X 0,Y 192.715,Z 416.475,A -85,B 0,C 180,E1 -21761.492,E2 -21761.492} C_VEL
LIN {X 0,Y 192.755,Z 416.475,A -85,B 0,C 180,E1 -21765.211,E2 -21765.211} C_VEL
LIN {X 0,Y 192.966,Z 416.443,A -85,B 0,C 180,E1 -21769.566,E2 -21769.566} C_VEL
LIN {X 0,Y 192.994,Z 416.443,A -85,B 0,C 180,E1 -21773.726,E2 -21773.726} C_VEL
LIN {X 0,Y 193.276,Z 416.405,A -85,B 0,C 180,E1 -21777.914,E2 -21777.914} C_VEL
LIN {X 0,Y 193.449,Z 416.385,A -85,B 0,C 180,E1 -21779.998,E2 -21779.998} C_VEL
LIN {X 0,Y 192.958,Z 416.448,A -85,B 0,C 180,E1 -21784.176,E2 -21784.176} C_VEL
LIN {X 0,Y 193.039,Z 416.436,A -85,B 0,C 180,E1 -21788.372,E2 -21788.372} C_VEL
LIN {X 0,Y 192.807,Z 416.469,A -85,B 0,C 180,E1 -21792.631,E2 -21792.631} C_VEL
LIN {X 0,Y 192.732,Z 416.478,A -85,B 0,C 180,E1 -21796.959,E2 -21796.959} C_VEL
LIN {X 0,Y 192.598,Z 416.491,A -85,B 0,C 180,E1 -21801.4,E2 -21801.4} C_VEL
LIN {X 0,Y 192.655,Z 416.482,A -85,B 0,C 180,E1 -21804.204,E2 -21804.204} C_VEL
LIN {X 0,Y 192.651,Z 416.487,A -85,B 0,C 180,E1 -21808.88,E2 -21808.88} C_VEL
LIN {X 0,Y 192.608,Z 416.491,A -85,B 0,C 180,E1 -21813.182,E2 -21813.182} C_VEL
LIN {X 0,Y 192.562,Z 416.498,A -85,B 0,C 180,E1 -21818.347,E2 -21818.347} C_VEL
LIN {X 0,Y 192.5,Z 416.505,A -85,B 0,C 180,E1 -21823.089,E2 -21823.089} C_VEL
LIN {X 0,Y 192.497,Z 416.504,A -85,B 0,C 180,E1 -21826.9,E2 -21826.9} C_VEL
LIN {X 0,Y 192.553,Z 416.498,A -85,B 0,C 180,E1 -21831.64,E2 -21831.64} C_VEL
LIN {X 0,Y 192.603,Z 416.49,A -85,B 0,C 180,E1 -21836.807,E2 -21836.807} C_VEL
LIN {X 0,Y 192.67,Z 416.484,A -85,B 0,C 180,E1 -21841.685,E2 -21841.685} C_VEL
LIN {X 0,Y 192.709,Z 416.478,A -85,B 0,C 180,E1 -21846.342,E2 -21846.342} C_VEL
LIN {X 0,Y 192.734,Z 416.475,A -85,B 0,C 180,E1 -21851.45,E2 -21851.45} C_VEL
LIN {X 0,Y 192.764,Z 416.47,A -85,B 0,C 180,E1 -21855.206,E2 -21855.206} C_VEL
LIN {X 0,Y 192.943,Z 416.449,A -85,B 0,C 180,E1 -21859.559,E2 -21859.559} C_VEL
LIN {X 0,Y 192.981,Z 416.443,A -85,B 0,C 180,E1 -21863.72,E2 -21863.72} C_VEL
LIN {X 0,Y 193.257,Z 416.412,A -85,B 0,C 180,E1 -21867.908,E2 -21867.908} C_VEL
LIN {X 0,Y 193.437,Z 416.387,A -85,B 0,C 180,E1 -21869.992,E2 -21869.992} C_VEL
LIN {X 0,Y 192.972,Z 416.449,A -85,B 0,C 180,E1 -21874.169,E2 -21874.169} C_VEL
LIN {X 0,Y 193.069,Z 416.432,A -85,B 0,C 180,E1 -21878.364,E2 -21878.364} C_VEL
LIN {X 0,Y 192.842,Z 416.463,A -85,B 0,C 180,E1 -21882.622,E2 -21882.622} C_VEL
LIN {X 0,Y 192.744,Z 416.47,A -85,B 0,C 180,E1 -21886.951,E2 -21886.951} C_VEL
LIN {X 0,Y 192.577,Z 416.496,A -85,B 0,C 180,E1 -21891.395,E2 -21891.395} C_VEL
LIN {X 0,Y 192.548,Z 416.5,A -85,B 0,C 180,E1 -21894.152,E2 -21894.152} C_VEL
LIN {X 0,Y 192.185,Z 416.545,A -85,B 0,C 180,E1 -21898.644,E2 -21898.644} C_VEL
LIN {X 0,Y 191.801,Z 416.643,A -85,B 0,C 180,E1 -21902.316,E2 -21902.316} C_VEL
LIN {X 0,Y 195.013,Z 428.681,A -85,B 0,C 180,E1 -21903.731,E2 -21903.731} C_VEL
LIN {X 0,Y 197.438,Z 440.169,A -85,B 0,C 180,E1 -21905.33,E2 -21905.33} C_VEL
LIN {X 0,Y 199.376,Z 451.05,A -85,B 0,C 180,E1 -21907.122,E2 -21907.122} C_VEL
LIN {X 0,Y 199.837,Z 453.922,A -85,B 0,C 180,E1 -21907.655,E2 -21907.655} C_VEL
LIN {X 0,Y 198.808,Z 461.164,A -85,B 0,C 180,E1 -21908.951,E2 -21908.951} C_VEL
LIN {X 0,Y 196.82,Z 472.572,A -85,B 0,C 180,E1 -21911.425,E2 -21911.425} C_VEL
LIN {X 0,Y 195.108,Z 481.864,A -85,B 0,C 180,E1 -21913.914,E2 -21913.914} C_VEL
LIN {X 0,Y 193.356,Z 491.466,A -85,B 0,C 180,E1 -21917.125,E2 -21917.125} C_VEL
LIN {X 0,Y 192.158,Z 498.755,A -85,B 0,C 180,E1 -21920.165,E2 -21920.165} C_VEL
LIN {X 0,Y 191.226,Z 504.875,A -85,B 0,C 180,E1 -21923.331,E2 -21923.331} C_VEL
LIN {X 0,Y 190.692,Z 509.652,A -85,B 0,C 180,E1 -21926.441,E2 -21926.441} C_VEL
LIN {X 0,Y 190.233,Z 513.927,A -85,B 0,C 180,E1 -21930.085,E2 -21930.085} C_VEL
LIN {X 0,Y 190.288,Z 516.847,A -85,B 0,C 180,E1 -21933.694,E2 -21933.694} C_VEL
LIN {X 0,Y 190.825,Z 518.528,A -85,B 0,C 180,E1 -21937.01,E2 -21937.01} C_VEL
LIN {X 0,Y 191.971,Z 519.273,A -85,B 0,C 180,E1 -21940.764,E2 -21940.764} C_VEL
LIN {X 0,Y 193.013,Z 519.129,A -85,B 0,C 180,E1 -21943.066,E2 -21943.066} C_VEL
LIN {X 0,Y 195.099,Z 518.032,A -85,B 0,C 180,E1 -21946.519,E2 -21946.519} C_VEL
LIN {X 0,Y 197.618,Z 515.981,A -85,B 0,C 180,E1 -21949.759,E2 -21949.759} C_VEL
LIN {X 0,Y 200.734,Z 512.846,A -85,B 0,C 180,E1 -21952.963,E2 -21952.963} C_VEL
LIN {X 0,Y 204.568,Z 508.521,A -85,B 0,C 180,E1 -21956.062,E2 -21956.062} C_VEL
LIN {X 0,Y 208.939,Z 502.986,A -85,B 0,C 180,E1 -21959.038,E2 -21959.038} C_VEL
LIN {X 0,Y 213.771,Z 495.998,A -85,B 0,C 180,E1 -21961.886,E2 -21961.886} C_VEL
LIN {X 0,Y 219.095,Z 487.509,A -85,B 0,C 180,E1 -21964.51,E2 -21964.51} C_VEL
LIN {X 0,Y 221.211,Z 483.828,A -85,B 0,C 180,E1 -21965.471,E2 -21965.471} C_VEL
LIN {X 0,Y 221.712,Z 481.927,A -85,B 0,C 180,E1 -21966.143,E2 -21966.143} C_VEL
LIN {X 0,Y 222.126,Z 474.651,A -85,B 0,C 180,E1 -21969.104,E2 -21969.104} C_VEL
LIN {X 0,Y 221.374,Z 468.478,A -85,B 0,C 180,E1 -21972.078,E2 -21972.078} C_VEL
LIN {X 0,Y 220.652,Z 465.472,A -85,B 0,C 180,E1 -21973.762,E2 -21973.762} C_VEL
LIN {X 0,Y 219.053,Z 461.116,A -85,B 0,C 180,E1 -21976.785,E2 -21976.785} C_VEL
LIN {X 0,Y 218.053,Z 458.822,A -85,B 0,C 180,E1 -21978.804,E2 -21978.804} C_VEL
LIN {X 0,Y 216.19,Z 455.547,A -85,B 0,C 180,E1 -21982.962,E2 -21982.962} C_VEL
LIN {X 0,Y 215.515,Z 454.57,A -85,B 0,C 180,E1 -21985.085,E2 -21985.085} C_VEL
LIN {X 0,Y 214.522,Z 454.507,A -85,B 0,C 180,E1 -21989.436,E2 -21989.436} C_VEL
LIN {X 0,Y 214.483,Z 455.039,A -85,B 0,C 180,E1 -21991.621,E2 -21991.621} C_VEL
LIN {X 0,Y 215.242,Z 457.293,A -85,B 0,C 180,E1 -21995.998,E2 -21995.998} C_VEL
LIN {X 0,Y 216.017,Z 459.096,A -85,B 0,C 180,E1 -21998.183,E2 -21998.183} C_VEL
LIN {X 0,Y 217.762,Z 465.206,A -85,B 0,C 180,E1 -22002.67,E2 -22002.67} C_VEL
LIN {X 0,Y 218.966,Z 470.54,A -85,B 0,C 180,E1 -22005.543,E2 -22005.543} C_VEL
LIN {X 0,Y 219.549,Z 474.703,A -85,B 0,C 180,E1 -22007.415,E2 -22007.415} C_VEL
LIN {X 0,Y 219.276,Z 480.885,A -85,B 0,C 180,E1 -22009.516,E2 -22009.516} C_VEL
LIN {X 0,Y 218.255,Z 489.43,A -85,B 0,C 180,E1 -22012.289,E2 -22012.289} C_VEL
LIN {X 0,Y 216.401,Z 497.576,A -85,B 0,C 180,E1 -22014.832,E2 -22014.832} C_VEL
LIN {X 0,Y 213.909,Z 504.912,A -85,B 0,C 180,E1 -22017.182,E2 -22017.182} C_VEL
LIN {X 0,Y 211.779,Z 509.079,A -85,B 0,C 180,E1 -22018.498,E2 -22018.498} C_VEL
LIN {X 0,Y 206.304,Z 517.567,A -85,B 0,C 180,E1 -22021.524,E2 -22021.524} C_VEL
LIN {X 0,Y 202.127,Z 523.504,A -85,B 0,C 180,E1 -22024.247,E2 -22024.247} C_VEL
LIN {X 0,Y 198.719,Z 528.374,A -85,B 0,C 180,E1 -22027.115,E2 -22027.115} C_VEL
LIN {X 0,Y 195.14,Z 533.364,A -85,B 0,C 180,E1 -22031.095,E2 -22031.095} C_VEL
LIN {X 0,Y 192.406,Z 536.675,A -85,B 0,C 180,E1 -22035.122,E2 -22035.122} C_VEL
LIN {X 0,Y 190.954,Z 537.693,A -85,B 0,C 180,E1 -22036.809,E2 -22036.809} C_VEL
LIN {X 0,Y 187.264,Z 538.555,A -85,B 0,C 180,E1 -22039.587,E2 -22039.587} C_VEL
LIN {X 0,Y 184.528,Z 538.67,A -85,B 0,C 180,E1 -22041.892,E2 -22041.892} C_VEL
LIN {X 0,Y 183.415,Z 538.475,A -85,B 0,C 180,E1 -22043.705,E2 -22043.705} C_VEL
LIN {X 0,Y 183.335,Z 538.333,A -85,B 0,C 180,E1 -22044.322,E2 -22044.322} C_VEL
LIN {X 0,Y 183.497,Z 537.238,A -85,B 0,C 180,E1 -22047.813,E2 -22047.813} C_VEL
LIN {X 0,Y 183.642,Z 535.985,A -85,B 0,C 180,E1 -22050.008,E2 -22050.008} C_VEL
LIN {X 0,Y 183.62,Z 533.226,A -85,B 0,C 180,E1 -22053.299,E2 -22053.299} C_VEL
LIN {X 0,Y 183.677,Z 529.356,A -85,B 0,C 180,E1 -22056.599,E2 -22056.599} C_VEL
LIN {X 0,Y 183.971,Z 524.278,A -85,B 0,C 180,E1 -22059.907,E2 -22059.907} C_VEL
LIN {X 0,Y 184.7,Z 517.851,A -85,B 0,C 180,E1 -22063.205,E2 -22063.205} C_VEL
LIN {X 0,Y 186.034,Z 509.892,A -85,B 0,C 180,E1 -22066.467,E2 -22066.467} C_VEL
LIN {X 0,Y 187.315,Z 501.738,A -85,B 0,C 180,E1 -22069.173,E2 -22069.173} C_VEL
LIN {X 0,Y 189.38,Z 491.502,A -85,B 0,C 180,E1 -22071.907,E2 -22071.907} C_VEL
LIN {X 0,Y 189.847,Z 488.691,A -85,B 0,C 180,E1 -22072.564,E2 -22072.564} C_VEL
LIN {X 0,Y 189.354,Z 477.191,A -85,B 0,C 180,E1 -22074.981,E2 -22074.981} C_VEL
LIN {X 0,Y 188.527,Z 464.391,A -85,B 0,C 180,E1 -22077.179,E2 -22077.179} C_VEL
LIN {X 0,Y 187.515,Z 452.137,A -85,B 0,C 180,E1 -22078.86,E2 -22078.86} C_VEL
LIN {X 0,Y 186.105,Z 437.689,A -85,B 0,C 180,E1 -22080.387,E2 -22080.387} C_VEL
LIN {X 0,Y 185.775,Z 434.275,A -85,B 0,C 180,E1 -22080.718,E2 -22080.718} C_VEL
LIN {X 0,Y 187.143,Z 429.705,A -85,B 0,C 180,E1 -22085.606,E2 -22085.606} C_VEL
LIN {X 0,Y 187.508,Z 427.441,A -85,B 0,C 180,E1 -22088.082,E2 -22088.082} C_VEL
LIN {X 0,Y 187.08,Z 424.631,A -85,B 0,C 180,E1 -22091.291,E2 -22091.291} C_VEL
LIN {X 0,Y 186.298,Z 420.831,A -85,B 0,C 180,E1 -22095.798,E2 -22095.798} C_VEL
LIN {X 0,Y 185.644,Z 417.359,A -85,B 0,C 180,E1 -22100.292,E2 -22100.292} C_VEL
LIN {X 0,Y 185.518,Z 417.373,A -85,B 0,C 180,E1 -22105.37,E2 -22105.37} C_VEL
LIN {X 0,Y 185.564,Z 417.369,A -85,B 0,C 180,E1 -22110.502,E2 -22110.502} C_VEL
LIN {X 0,Y 185.602,Z 417.365,A -85,B 0,C 180,E1 -22115.383,E2 -22115.383} C_VEL
LIN {X 0,Y 185.646,Z 417.356,A -85,B 0,C 180,E1 -22121.179,E2 -22121.179} C_VEL
LIN {X 0,Y 185.685,Z 417.354,A -85,B 0,C 180,E1 -22124.635,E2 -22124.635} C_VEL
LIN {X 0,Y 185.909,Z 417.322,A -85,B 0,C 180,E1 -22129.418,E2 -22129.418} C_VEL
LIN {X 0,Y 185.957,Z 417.321,A -85,B 0,C 180,E1 -22133.488,E2 -22133.488} C_VEL
LIN {X 0,Y 186.22,Z 417.283,A -85,B 0,C 180,E1 -22137.835,E2 -22137.835} C_VEL
LIN {X 0,Y 186.413,Z 417.261,A -85,B 0,C 180,E1 -22139.998,E2 -22139.998} C_VEL
LIN {X 0,Y 185.906,Z 417.327,A -85,B 0,C 180,E1 -22144.334,E2 -22144.334} C_VEL
LIN {X 0,Y 185.99,Z 417.316,A -85,B 0,C 180,E1 -22148.691,E2 -22148.691} C_VEL
LIN {X 0,Y 185.732,Z 417.347,A -85,B 0,C 180,E1 -22153.121,E2 -22153.121} C_VEL
LIN {X 0,Y 185.669,Z 417.355,A -85,B 0,C 180,E1 -22157.625,E2 -22157.625} C_VEL
LIN {X 0,Y 185.57,Z 417.367,A -85,B 0,C 180,E1 -22162.252,E2 -22162.252} C_VEL
LIN {X 0,Y 185.568,Z 417.37,A -85,B 0,C 180,E1 -22167.029,E2 -22167.029} C_VEL
LIN {X 0,Y 185.591,Z 417.365,A -85,B 0,C 180,E1 -22169.489,E2 -22169.489} C_VEL
LIN {X 0,Y 185.511,Z 417.377,A -85,B 0,C 180,E1 -22174.627,E2 -22174.627} C_VEL
LIN {X 0,Y 185.517,Z 417.374,A -85,B 0,C 180,E1 -22177.308,E2 -22177.308} C_VEL
LIN {X 0,Y 185.481,Z 417.378,A -85,B 0,C 180,E1 -22180.718,E2 -22180.718} C_VEL
LIN {X 0,Y 185.467,Z 417.382,A -85,B 0,C 180,E1 -22186.049,E2 -22186.049} C_VEL
LIN {X 0,Y 185.468,Z 417.378,A -85,B 0,C 180,E1 -22189.886,E2 -22189.886} C_VEL
LIN {X 0,Y 185.51,Z 417.377,A -85,B 0,C 180,E1 -22192.706,E2 -22192.706} C_VEL
LIN {X 0,Y 185.549,Z 417.368,A -85,B 0,C 180,E1 -22197.968,E2 -22197.968} C_VEL
LIN {X 0,Y 185.587,Z 417.368,A -85,B 0,C 180,E1 -22200.569,E2 -22200.569} C_VEL
LIN {X 0,Y 185.591,Z 417.361,A -85,B 0,C 180,E1 -22205.375,E2 -22205.375} C_VEL
LIN {X 0,Y 185.609,Z 417.365,A -85,B 0,C 180,E1 -22210.068,E2 -22210.068} C_VEL
LIN {X 0,Y 185.695,Z 417.352,A -85,B 0,C 180,E1 -22214.63,E2 -22214.63} C_VEL
LIN {X 0,Y 185.887,Z 417.328,A -85,B 0,C 180,E1 -22219.41,E2 -22219.41} C_VEL
LIN {X 0,Y 185.944,Z 417.319,A -85,B 0,C 180,E1 -22223.482,E2 -22223.482} C_VEL
LIN {X 0,Y 186.201,Z 417.291,A -85,B 0,C 180,E1 -22227.829,E2 -22227.829} C_VEL
LIN {X 0,Y 186.4,Z 417.263,A -85,B 0,C 180,E1 -22229.992,E2 -22229.992} C_VEL
LIN {X 0,Y 185.919,Z 417.327,A -85,B 0,C 180,E1 -22234.328,E2 -22234.328} C_VEL
LIN {X 0,Y 186.019,Z 417.309,A -85,B 0,C 180,E1 -22238.684,E2 -22238.684} C_VEL
LIN {X 0,Y 185.753,Z 417.345,A -85,B 0,C 180,E1 -22243.113,E2 -22243.113} C_VEL
LIN {X 0,Y 185.676,Z 417.351,A -85,B 0,C 180,E1 -22247.617,E2 -22247.617} C_VEL
LIN {X 0,Y 185.52,Z 417.375,A -85,B 0,C 180,E1 -22252.252,E2 -22252.252} C_VEL
LIN {X 0,Y 185.455,Z 417.382,A -85,B 0,C 180,E1 -22254.627,E2 -22254.627} C_VEL
LIN {X 0,Y 184.992,Z 417.442,A -85,B 0,C 180,E1 -22259.586,E2 -22259.586} C_VEL
LIN {X 0,Y 184.833,Z 417.463,A -85,B 0,C 180,E1 -22261.671,E2 -22261.671} C_VEL
LIN {X 0,Y 188.327,Z 430.637,A -85,B 0,C 180,E1 -22263.345,E2 -22263.345} C_VEL
LIN {X 0,Y 190.853,Z 443.061,A -85,B 0,C 180,E1 -22265.212,E2 -22265.212} C_VEL
LIN {X 0,Y 192.761,Z 454.165,A -85,B 0,C 180,E1 -22267.202,E2 -22267.202} C_VEL
LIN {X 0,Y 192.559,Z 457.367,A -85,B 0,C 180,E1 -22267.787,E2 -22267.787} C_VEL
LIN {X 0,Y 190.514,Z 468.812,A -85,B 0,C 180,E1 -22270.137,E2 -22270.137} C_VEL
LIN {X 0,Y 188.742,Z 478.695,A -85,B 0,C 180,E1 -22272.661,E2 -22272.661} C_VEL
LIN {X 0,Y 186.981,Z 487.854,A -85,B 0,C 180,E1 -22275.56,E2 -22275.56} C_VEL
LIN {X 0,Y 185.459,Z 496.37,A -85,B 0,C 180,E1 -22278.909,E2 -22278.909} C_VEL
LIN {X 0,Y 184.353,Z 503.457,A -85,B 0,C 180,E1 -22282.416,E2 -22282.416} C_VEL
LIN {X 0,Y 183.627,Z 509.474,A -85,B 0,C 180,E1 -22286.296,E2 -22286.296} C_VEL
LIN {X 0,Y 183.133,Z 513.883,A -85,B 0,C 180,E1 -22290.076,E2 -22290.076} C_VEL
LIN {X 0,Y 183.102,Z 516.086,A -85,B 0,C 180,E1 -22292.577,E2 -22292.577} C_VEL
LIN {X 0,Y 183.637,Z 518.549,A -85,B 0,C 180,E1 -22296.684,E2 -22296.684} C_VEL
LIN {X 0,Y 184.552,Z 519.56,A -85,B 0,C 180,E1 -22299.959,E2 -22299.959} C_VEL
LIN {X 0,Y 185.526,Z 519.755,A -85,B 0,C 180,E1 -22302.361,E2 -22302.361} C_VEL
LIN {X 0,Y 187.893,Z 519.014,A -85,B 0,C 180,E1 -22306.494,E2 -22306.494} C_VEL
LIN {X 0,Y 190.023,Z 517.61,A -85,B 0,C 180,E1 -22309.345,E2 -22309.345} C_VEL
LIN {X 0,Y 193.096,Z 515.009,A -85,B 0,C 180,E1 -22312.683,E2 -22312.683} C_VEL
LIN {X 0,Y 197.204,Z 511.025,A -85,B 0,C 180,E1 -22316.12,E2 -22316.12} C_VEL
LIN {X 0,Y 201.293,Z 506.416,A -85,B 0,C 180,E1 -22319.002,E2 -22319.002} C_VEL
LIN {X 0,Y 206.266,Z 500.128,A -85,B 0,C 180,E1 -22321.954,E2 -22321.954} C_VEL
LIN {X 0,Y 211.5,Z 492.739,A -85,B 0,C 180,E1 -22324.637,E2 -22324.637} C_VEL
LIN {X 0,Y 215.761,Z 486.076,A -85,B 0,C 180,E1 -22326.548,E2 -22326.548} C_VEL
LIN {X 0,Y 216.548,Z 481.654,A -85,B 0,C 180,E1 -22328.399,E2 -22328.399} C_VEL
LIN {X 0,Y 216.825,Z 478.33,A -85,B 0,C 180,E1 -22329.92,E2 -22329.92} C_VEL
LIN {X 0,Y 216.36,Z 472.264,A -85,B 0,C 180,E1 -22333.145,E2 -22333.145} C_VEL
LIN {X 0,Y 215.327,Z 468.395,A -85,B 0,C 180,E1 -22335.8,E2 -22335.8} C_VEL
LIN {X 0,Y 214.393,Z 465.654,A -85,B 0,C 180,E1 -22338.103,E2 -22338.103} C_VEL
LIN {X 0,Y 213.994,Z 464.52,A -85,B 0,C 180,E1 -22339.175,E2 -22339.175} C_VEL
LIN {X 0,Y 212.481,Z 461.476,A -85,B 0,C 180,E1 -22343.387,E2 -22343.387} C_VEL
LIN {X 0,Y 211.638,Z 460.681,A -85,B 0,C 180,E1 -22346.304,E2 -22346.304} C_VEL
LIN {X 0,Y 211.066,Z 460.875,A -85,B 0,C 180,E1 -22350.05,E2 -22350.05} C_VEL
LIN {X 0,Y 211.373,Z 462.585,A -85,B 0,C 180,E1 -22354.421,E2 -22354.421} C_VEL
LIN {X 0,Y 212.109,Z 464.604,A -85,B 0,C 180,E1 -22357.338,E2 -22357.338} C_VEL
LIN {X 0,Y 213.496,Z 470.293,A -85,B 0,C 180,E1 -22361.956,E2 -22361.956} C_VEL
LIN {X 0,Y 214.528,Z 476.405,A -85,B 0,C 180,E1 -22365.443,E2 -22365.443} C_VEL
LIN {X 0,Y 214.651,Z 480.074,A -85,B 0,C 180,E1 -22367.084,E2 -22367.084} C_VEL
LIN {X 0,Y 213.474,Z 488.546,A -85,B 0,C 180,E1 -22370.08,E2 -22370.08} C_VEL
LIN {X 0,Y 212.106,Z 494.739,A -85,B 0,C 180,E1 -22372.206,E2 -22372.206} C_VEL
LIN {X 0,Y 209.694,Z 502.464,A -85,B 0,C 180,E1 -22374.818,E2 -22374.818} C_VEL
LIN {X 0,Y 206.704,Z 508.953,A -85,B 0,C 180,E1 -22377.053,E2 -22377.053} C_VEL
LIN {X 0,Y 200.941,Z 517.349,A -85,B 0,C 180,E1 -22380.115,E2 -22380.115} C_VEL
LIN {X 0,Y 195.788,Z 524.131,A -85,B 0,C 180,E1 -22383.349,E2 -22383.349} C_VEL
LIN {X 0,Y 192.184,Z 528.74,A -85,B 0,C 180,E1 -22386.29,E2 -22386.29} C_VEL
LIN {X 0,Y 188.409,Z 533.43,A -85,B 0,C 180,E1 -22390.393,E2 -22390.393} C_VEL
LIN {X 0,Y 185.483,Z 536.597,A -85,B 0,C 180,E1 -22394.628,E2 -22394.628} C_VEL
LIN {X 0,Y 183.918,Z 538.298,A -85,B 0,C 180,E1 -22398.994,E2 -22398.994} C_VEL
LIN {X 0,Y 183.347,Z 538.504,A -85,B 0,C 180,E1 -22403.405,E2 -22403.405} C_VEL
LIN {X 0,Y 183.335,Z 538.333,A -85,B 0,C 180,E1 -22404.322,E2 -22404.322} C_VEL
LIN {X 0,Y 183.04,Z 538.047,A -85,B 0,C 180,E1 -22405.545,E2 -22405.545} C_VEL
LIN {X 0,Y 181.744,Z 537.256,A -85,B 0,C 180,E1 -22407.346,E2 -22407.346} C_VEL
LIN {X 0,Y 178.686,Z 535.17,A -85,B 0,C 180,E1 -22410.302,E2 -22410.302} C_VEL
LIN {X 0,Y 176.848,Z 532.942,A -85,B 0,C 180,E1 -22412.724,E2 -22412.724} C_VEL
LIN {X 0,Y 176.595,Z 531.65,A -85,B 0,C 180,E1 -22413.958,E2 -22413.958} C_VEL
LIN {X 0,Y 176.649,Z 528.172,A -85,B 0,C 180,E1 -22416.863,E2 -22416.863} C_VEL
LIN {X 0,Y 177.092,Z 521.936,A -85,B 0,C 180,E1 -22420.874,E2 -22420.874} C_VEL
LIN {X 0,Y 177.975,Z 515.064,A -85,B 0,C 180,E1 -22424.297,E2 -22424.297} C_VEL
LIN {X 0,Y 179.424,Z 506.481,A -85,B 0,C 180,E1 -22427.68,E2 -22427.68} C_VEL
LIN {X 0,Y 181.027,Z 497.753,A -85,B 0,C 180,E1 -22430.459,E2 -22430.459} C_VEL
LIN {X 0,Y 182.701,Z 489.445,A -85,B 0,C 180,E1 -22432.631,E2 -22432.631} C_VEL
LIN {X 0,Y 182.369,Z 478.529,A -85,B 0,C 180,E1 -22435.09,E2 -22435.09} C_VEL
LIN {X 0,Y 181.609,Z 465.751,A -85,B 0,C 180,E1 -22437.431,E2 -22437.431} C_VEL
LIN {X 0,Y 180.672,Z 453.625,A -85,B 0,C 180,E1 -22439.234,E2 -22439.234} C_VEL
LIN {X 0,Y 179.417,Z 439.854,A -85,B 0,C 180,E1 -22440.821,E2 -22440.821} C_VEL
LIN {X 0,Y 178.828,Z 433.904,A -85,B 0,C 180,E1 -22441.414,E2 -22441.414} C_VEL
LIN {X 0,Y 180.085,Z 429.95,A -85,B 0,C 180,E1 -22445.839,E2 -22445.839} C_VEL
LIN {X 0,Y 180.346,Z 427.363,A -85,B 0,C 180,E1 -22448.792,E2 -22448.792} C_VEL
LIN {X 0,Y 179.6,Z 423.397,A -85,B 0,C 180,E1 -22453.564,E2 -22453.564} C_VEL
LIN {X 0,Y 178.696,Z 418.718,A -85,B 0,C 180,E1 -22459.536,E2 -22459.536} C_VEL
LIN {X 0,Y 178.614,Z 418.234,A -85,B 0,C 180,E1 -22460.251,E2 -22460.251} C_VEL
LIN {X 0,Y 178.504,Z 418.246,A -85,B 0,C 180,E1 -22466.548,E2 -22466.548} C_VEL
LIN {X 0,Y 178.463,Z 418.251,A -85,B 0,C 180,E1 -22471.797,E2 -22471.797} C_VEL
LIN {X 0,Y 178.537,Z 418.243,A -85,B 0,C 180,E1 -22474.89,E2 -22474.89} C_VEL
LIN {X 0,Y 178.628,Z 418.229,A -85,B 0,C 180,E1 -22481.652,E2 -22481.652} C_VEL
LIN {X 0,Y 178.662,Z 418.229,A -85,B 0,C 180,E1 -22486.346,E2 -22486.346} C_VEL
LIN {X 0,Y 178.927,Z 418.194,A -85,B 0,C 180,E1 -22490.959,E2 -22490.959} C_VEL
LIN {X 0,Y 179.165,Z 418.162,A -85,B 0,C 180,E1 -22497.75,E2 -22497.75} C_VEL
LIN {X 0,Y 179.377,Z 418.138,A -85,B 0,C 180,E1 -22499.998,E2 -22499.998} C_VEL
LIN {X 0,Y 178.855,Z 418.206,A -85,B 0,C 180,E1 -22504.505,E2 -22504.505} C_VEL
LIN {X 0,Y 178.921,Z 418.198,A -85,B 0,C 180,E1 -22509.038,E2 -22509.038} C_VEL
LIN {X 0,Y 178.659,Z 418.227,A -85,B 0,C 180,E1 -22513.65,E2 -22513.65} C_VEL
LIN {X 0,Y 178.571,Z 418.241,A -85,B 0,C 180,E1 -22519.147,E2 -22519.147} C_VEL
LIN {X 0,Y 178.535,Z 418.244,A -85,B 0,C 180,E1 -22525.109,E2 -22525.109} C_VEL
LIN {X 0,Y 178.535,Z 418.244,A -85,B 0,C 180,E1 -22529.986,E2 -22529.986} C_VEL
LIN {X 0,Y 178.496,Z 418.249,A -85,B 0,C 180,E1 -22534.213,E2 -22534.213} C_VEL
LIN {X 0,Y 178.406,Z 418.258,A -85,B 0,C 180,E1 -22539.069,E2 -22539.069} C_VEL
LIN {X 0,Y 178.408,Z 418.259,A -85,B 0,C 180,E1 -22542.039,E2 -22542.039} C_VEL
LIN {X 0,Y 178.403,Z 418.261,A -85,B 0,C 180,E1 -22545.158,E2 -22545.158} C_VEL
LIN {X 0,Y 178.408,Z 418.258,A -85,B 0,C 180,E1 -22548.454,E2 -22548.454} C_VEL
LIN {X 0,Y 178.428,Z 418.258,A -85,B 0,C 180,E1 -22553.775,E2 -22553.775} C_VEL
LIN {X 0,Y 178.492,Z 418.247,A -85,B 0,C 180,E1 -22556.539,E2 -22556.539} C_VEL
LIN {X 0,Y 178.528,Z 418.246,A -85,B 0,C 180,E1 -22559.999,E2 -22559.999} C_VEL
LIN {X 0,Y 178.539,Z 418.24,A -85,B 0,C 180,E1 -22564.868,E2 -22564.868} C_VEL
LIN {X 0,Y 178.625,Z 418.233,A -85,B 0,C 180,E1 -22570.776,E2 -22570.776} C_VEL
LIN {X 0,Y 178.658,Z 418.231,A -85,B 0,C 180,E1 -22576.34,E2 -22576.34} C_VEL
LIN {X 0,Y 178.909,Z 418.195,A -85,B 0,C 180,E1 -22580.952,E2 -22580.952} C_VEL
LIN {X 0,Y 179.147,Z 418.169,A -85,B 0,C 180,E1 -22587.744,E2 -22587.744} C_VEL
LIN {X 0,Y 179.363,Z 418.139,A -85,B 0,C 180,E1 -22589.992,E2 -22589.992} C_VEL
LIN {X 0,Y 178.868,Z 418.204,A -85,B 0,C 180,E1 -22594.499,E2 -22594.499} C_VEL
LIN {X 0,Y 178.968,Z 418.186,A -85,B 0,C 180,E1 -22599.029,E2 -22599.029} C_VEL
LIN {X 0,Y 178.675,Z 418.228,A -85,B 0,C 180,E1 -22603.642,E2 -22603.642} C_VEL
LIN {X 0,Y 178.635,Z 418.232,A -85,B 0,C 180,E1 -22608.336,E2 -22608.336} C_VEL
LIN {X 0,Y 178.41,Z 418.259,A -85,B 0,C 180,E1 -22613.189,E2 -22613.189} C_VEL
LIN {X 0,Y 178.283,Z 418.277,A -85,B 0,C 180,E1 -22615.688,E2 -22615.688} C_VEL
LIN {X 0,Y 177.833,Z 418.345,A -85,B 0,C 180,E1 -22621.069,E2 -22621.069} C_VEL
LIN {X 0,Y 181.468,Z 431.733,A -85,B 0,C 180,E1 -22622.823,E2 -22622.823} C_VEL
LIN {X 0,Y 183.805,Z 443.361,A -85,B 0,C 180,E1 -22624.653,E2 -22624.653} C_VEL
LIN {X 0,Y 185.852,Z 455.841,A -85,B 0,C 180,E1 -22626.998,E2 -22626.998} C_VEL
LIN {X 0,Y 183.874,Z 467.073,A -85,B 0,C 180,E1 -22629.29,E2 -22629.29} C_VEL
LIN {X 0,Y 181.965,Z 477.653,A -85,B 0,C 180,E1 -22632.003,E2 -22632.003} C_VEL
LIN {X 0,Y 180.125,Z 486.903,A -85,B 0,C 180,E1 -22634.934,E2 -22634.934} C_VEL
LIN {X 0,Y 178.517,Z 495.614,A -85,B 0,C 180,E1 -22638.404,E2 -22638.404} C_VEL
LIN {X 0,Y 177.425,Z 502.25,A -85,B 0,C 180,E1 -22641.689,E2 -22641.689} C_VEL
LIN {X 0,Y 176.722,Z 507.338,A -85,B 0,C 180,E1 -22644.788,E2 -22644.788} C_VEL
LIN {X 0,Y 176.158,Z 512.461,A -85,B 0,C 180,E1 -22648.761,E2 -22648.761} C_VEL
LIN {X 0,Y 175.997,Z 515.124,A -85,B 0,C 180,E1 -22651.443,E2 -22651.443} C_VEL
LIN {X 0,Y 176.1,Z 517.086,A -85,B 0,C 180,E1 -22653.962,E2 -22653.962} C_VEL
LIN {X 0,Y 176.513,Z 518.614,A -85,B 0,C 180,E1 -22656.539,E2 -22656.539} C_VEL
LIN {X 0,Y 177.144,Z 519.598,A -85,B 0,C 180,E1 -22659.082,E2 -22659.082} C_VEL
LIN {X 0,Y 178.056,Z 520.138,A -85,B 0,C 180,E1 -22661.595,E2 -22661.595} C_VEL
LIN {X 0,Y 179.229,Z 520.232,A -85,B 0,C 180,E1 -22664.071,E2 -22664.071} C_VEL
LIN {X 0,Y 180.696,Z 519.825,A -85,B 0,C 180,E1 -22666.507,E2 -22666.507} C_VEL
LIN {X 0,Y 182.424,Z 518.998,A -85,B 0,C 180,E1 -22668.896,E2 -22668.896} C_VEL
LIN {X 0,Y 184.7,Z 517.527,A -85,B 0,C 180,E1 -22671.553,E2 -22671.553} C_VEL
LIN {X 0,Y 189.232,Z 513.802,A -85,B 0,C 180,E1 -22675.742,E2 -22675.742} C_VEL
LIN {X 0,Y 193.655,Z 509.509,A -85,B 0,C 180,E1 -22678.962,E2 -22678.962} C_VEL
LIN {X 0,Y 198.748,Z 503.97,A -85,B 0,C 180,E1 -22682.028,E2 -22682.028} C_VEL
LIN {X 0,Y 203.82,Z 497.635,A -85,B 0,C 180,E1 -22684.704,E2 -22684.704} C_VEL
LIN {X 0,Y 209.402,Z 489.813,A -85,B 0,C 180,E1 -22687.232,E2 -22687.232} C_VEL
LIN {X 0,Y 210.37,Z 488.325,A -85,B 0,C 180,E1 -22687.681,E2 -22687.681} C_VEL
LIN {X 0,Y 211.428,Z 483.058,A -85,B 0,C 180,E1 -22690.176,E2 -22690.176} C_VEL
LIN {X 0,Y 211.48,Z 478.43,A -85,B 0,C 180,E1 -22692.757,E2 -22692.757} C_VEL
LIN {X 0,Y 211.026,Z 475.015,A -85,B 0,C 180,E1 -22695.059,E2 -22695.059} C_VEL
LIN {X 0,Y 210.382,Z 472.023,A -85,B 0,C 180,E1 -22697.499,E2 -22697.499} C_VEL
LIN {X 0,Y 209.503,Z 469.681,A -85,B 0,C 180,E1 -22700.093,E2 -22700.093} C_VEL
LIN {X 0,Y 208.37,Z 467.124,A -85,B 0,C 180,E1 -22704.424,E2 -22704.424} C_VEL
LIN {X 0,Y 207.992,Z 466.741,A -85,B 0,C 180,E1 -22706.059,E2 -22706.059} C_VEL
LIN {X 0,Y 207.363,Z 467.107,A -85,B 0,C 180,E1 -22710.558,E2 -22710.558} C_VEL
LIN {X 0,Y 207.439,Z 467.909,A -85,B 0,C 180,E1 -22712.827,E2 -22712.827} C_VEL
LIN {X 0,Y 207.896,Z 469.556,A -85,B 0,C 180,E1 -22715.789,E2 -22715.789} C_VEL
LIN {X 0,Y 208.314,Z 471.602,A -85,B 0,C 180,E1 -22718.139,E2 -22718.139} C_VEL
LIN {X 0,Y 209.125,Z 475.658,A -85,B 0,C 180,E1 -22721.527,E2 -22721.527} C_VEL
LIN {X 0,Y 209.672,Z 480.918,A -85,B 0,C 180,E1 -22724.743,E2 -22724.743} C_VEL
LIN {X 0,Y 209.673,Z 483.84,A -85,B 0,C 180,E1 -22726.171,E2 -22726.171} C_VEL
LIN {X 0,Y 207.923,Z 492.371,A -85,B 0,C 180,E1 -22729.424,E2 -22729.424} C_VEL
LIN {X 0,Y 205.799,Z 499.64,A -85,B 0,C 180,E1 -22732.081,E2 -22732.081} C_VEL
LIN {X 0,Y 202.966,Z 506.399,A -85,B 0,C 180,E1 -22734.56,E2 -22734.56} C_VEL
LIN {X 0,Y 200.882,Z 510.233,A -85,B 0,C 180,E1 -22735.97,E2 -22735.97} C_VEL
LIN {X 0,Y 194.88,Z 518.248,A -85,B 0,C 180,E1 -22739.086,E2 -22739.086} C_VEL
LIN {X 0,Y 189.51,Z 524.666,A -85,B 0,C 180,E1 -22742.392,E2 -22742.392} C_VEL
LIN {X 0,Y 185.699,Z 529.078,A -85,B 0,C 180,E1 -22745.408,E2 -22745.408} C_VEL
LIN {X 0,Y 181.708,Z 533.507,A -85,B 0,C 180,E1 -22749.638,E2 -22749.638} C_VEL
LIN {X 0,Y 178.624,Z 536.449,A -85,B 0,C 180,E1 -22754.022,E2 -22754.022} C_VEL
LIN {X 0,Y 176.923,Z 537.909,A -85,B 0,C 180,E1 -22758.553,E2 -22758.553} C_VEL
LIN {X 0,Y 176.288,Z 537.954,A -85,B 0,C 180,E1 -22763.14,E2 -22763.14} C_VEL
LIN {X 0,Y 176.333,Z 537.425,A -85,B 0,C 180,E1 -22765.436,E2 -22765.436} C_VEL
LIN {X 0,Y 176.433,Z 536.47,A -85,B 0,C 180,E1 -22767.726,E2 -22767.726} C_VEL
LIN {X 0,Y 176.587,Z 535.105,A -85,B 0,C 180,E1 -22770.008,E2 -22770.008} C_VEL
LIN {X 0,Y 176.595,Z 531.65,A -85,B 0,C 180,E1 -22773.958,E2 -22773.958} C_VEL
LIN {X 0,Y 176.333,Z 530.297,A -85,B 0,C 180,E1 -22775.154,E2 -22775.154} C_VEL
LIN {X 0,Y 175.064,Z 527.975,A -85,B 0,C 180,E1 -22776.885,E2 -22776.885} C_VEL
LIN {X 0,Y 171.114,Z 521.513,A -85,B 0,C 180,E1 -22780.782,E2 -22780.782} C_VEL
LIN {X 0,Y 170.402,Z 518.354,A -85,B 0,C 180,E1 -22782.464,E2 -22782.464} C_VEL
LIN {X 0,Y 170.464,Z 517.244,A -85,B 0,C 180,E1 -22783.021,E2 -22783.021} C_VEL
LIN {X 0,Y 171.85,Z 509.169,A -85,B 0,C 180,E1 -22786.643,E2 -22786.643} C_VEL
LIN {X 0,Y 173.207,Z 501.09,A -85,B 0,C 180,E1 -22789.566,E2 -22789.566} C_VEL
LIN {X 0,Y 175.225,Z 491.612,A -85,B 0,C 180,E1 -22792.35,E2 -22792.35} C_VEL
LIN {X 0,Y 175.67,Z 487.767,A -85,B 0,C 180,E1 -22793.329,E2 -22793.329} C_VEL
LIN {X 0,Y 175.221,Z 476.617,A -85,B 0,C 180,E1 -22795.869,E2 -22795.869} C_VEL
LIN {X 0,Y 174.428,Z 463.251,A -85,B 0,C 180,E1 -22798.35,E2 -22798.35} C_VEL
LIN {X 0,Y 173.423,Z 450.28,A -85,B 0,C 180,E1 -22800.246,E2 -22800.246} C_VEL
LIN {X 0,Y 172.079,Z 436.04,A -85,B 0,C 180,E1 -22801.85,E2 -22801.85} C_VEL
LIN {X 0,Y 171.88,Z 433.537,A -85,B 0,C 180,E1 -22802.12,E2 -22802.12} C_VEL
LIN {X 0,Y 172.866,Z 430.555,A -85,B 0,C 180,E1 -22805.595,E2 -22805.595} C_VEL
LIN {X 0,Y 173.262,Z 428.959,A -85,B 0,C 180,E1 -22807.486,E2 -22807.486} C_VEL
LIN {X 0,Y 173.054,Z 426.468,A -85,B 0,C 180,E1 -22810.535,E2 -22810.535} C_VEL
LIN {X 0,Y 172.123,Z 422.174,A -85,B 0,C 180,E1 -22816.039,E2 -22816.039} C_VEL
LIN {X 0,Y 171.578,Z 419.111,A -85,B 0,C 180,E1 -22820.207,E2 -22820.207} C_VEL
LIN {X 0,Y 171.421,Z 419.128,A -85,B 0,C 180,E1 -22825.094,E2 -22825.094} C_VEL
LIN {X 0,Y 171.429,Z 419.13,A -85,B 0,C 180,E1 -22830.528,E2 -22830.528} C_VEL
LIN {X 0,Y 171.457,Z 419.126,A -85,B 0,C 180,E1 -22835.799,E2 -22835.799} C_VEL
LIN {X 0,Y 171.528,Z 419.116,A -85,B 0,C 180,E1 -22840.864,E2 -22840.864} C_VEL
LIN {X 0,Y 171.576,Z 419.112,A -85,B 0,C 180,E1 -22845.771,E2 -22845.771} C_VEL
LIN {X 0,Y 171.865,Z 419.071,A -85,B 0,C 180,E1 -22850.584,E2 -22850.584} C_VEL
LIN {X 0,Y 171.823,Z 419.081,A -85,B 0,C 180,E1 -22855.306,E2 -22855.306} C_VEL
LIN {X 0,Y 172.34,Z 419.014,A -85,B 0,C 180,E1 -22859.998,E2 -22859.998} C_VEL
LIN {X 0,Y 171.876,Z 419.072,A -85,B 0,C 180,E1 -22867.044,E2 -22867.044} C_VEL
LIN {X 0,Y 171.786,Z 419.088,A -85,B 0,C 180,E1 -22870.89,E2 -22870.89} C_VEL
LIN {X 0,Y 171.535,Z 419.115,A -85,B 0,C 180,E1 -22876.664,E2 -22876.664} C_VEL
LIN {X 0,Y 171.44,Z 419.127,A -85,B 0,C 180,E1 -22881.648,E2 -22881.648} C_VEL
LIN {X 0,Y 171.426,Z 419.133,A -85,B 0,C 180,E1 -22886.803,E2 -22886.803} C_VEL
LIN {X 0,Y 171.452,Z 419.126,A -85,B 0,C 180,E1 -22890.579,E2 -22890.579} C_VEL
LIN {X 0,Y 171.406,Z 419.134,A -85,B 0,C 180,E1 -22895.029,E2 -22895.029} C_VEL
LIN {X 0,Y 171.369,Z 419.135,A -85,B 0,C 180,E1 -22898.8,E2 -22898.8} C_VEL
LIN {X 0,Y 171.33,Z 419.143,A -85,B 0,C 180,E1 -22904.211,E2 -22904.211} C_VEL
LIN {X 0,Y 171.34,Z 419.138,A -85,B 0,C 180,E1 -22908.973,E2 -22908.973} C_VEL
LIN {X 0,Y 171.37,Z 419.138,A -85,B 0,C 180,E1 -22912.027,E2 -22912.027} C_VEL
LIN {X 0,Y 171.405,Z 419.131,A -85,B 0,C 180,E1 -22915.085,E2 -22915.085} C_VEL
LIN {X 0,Y 171.455,Z 419.129,A -85,B 0,C 180,E1 -22920.527,E2 -22920.527} C_VEL
LIN {X 0,Y 171.462,Z 419.121,A -85,B 0,C 180,E1 -22925.794,E2 -22925.794} C_VEL
LIN {X 0,Y 171.581,Z 419.11,A -85,B 0,C 180,E1 -22930.863,E2 -22930.863} C_VEL
LIN {X 0,Y 171.576,Z 419.11,A -85,B 0,C 180,E1 -22935.764,E2 -22935.764} C_VEL
LIN {X 0,Y 171.846,Z 419.076,A -85,B 0,C 180,E1 -22940.576,E2 -22940.576} C_VEL
LIN {X 0,Y 171.811,Z 419.082,A -85,B 0,C 180,E1 -22945.299,E2 -22945.299} C_VEL
LIN {X 0,Y 172.326,Z 419.016,A -85,B 0,C 180,E1 -22949.991,E2 -22949.991} C_VEL
LIN {X 0,Y 171.817,Z 419.082,A -85,B 0,C 180,E1 -22954.684,E2 -22954.684} C_VEL
LIN {X 0,Y 171.9,Z 419.067,A -85,B 0,C 180,E1 -22959.403,E2 -22959.403} C_VEL
LIN {X 0,Y 171.597,Z 419.11,A -85,B 0,C 180,E1 -22964.216,E2 -22964.216} C_VEL
LIN {X 0,Y 171.52,Z 419.118,A -85,B 0,C 180,E1 -22969.545,E2 -22969.545} C_VEL
LIN {X 0,Y 171.266,Z 419.15,A -85,B 0,C 180,E1 -22975.479,E2 -22975.479} C_VEL
LIN {X 0,Y 170.841,Z 419.225,A -85,B 0,C 180,E1 -22980.409,E2 -22980.409} C_VEL
LIN {X 0,Y 174.487,Z 432.364,A -85,B 0,C 180,E1 -22982.242,E2 -22982.242} C_VEL
LIN {X 0,Y 177.075,Z 445.54,A -85,B 0,C 180,E1 -22984.431,E2 -22984.431} C_VEL
LIN {X 0,Y 178.768,Z 455.931,A -85,B 0,C 180,E1 -22986.473,E2 -22986.473} C_VEL
LIN {X 0,Y 178.072,Z 461.177,A -85,B 0,C 180,E1 -22987.53,E2 -22987.53} C_VEL
LIN {X 0,Y 176.03,Z 472.03,A -85,B 0,C 180,E1 -22990.076,E2 -22990.076} C_VEL
LIN {X 0,Y 174.072,Z 481.923,A -85,B 0,C 180,E1 -22992.967,E2 -22992.967} C_VEL
LIN {X 0,Y 172.336,Z 490.663,A -85,B 0,C 180,E1 -22996.113,E2 -22996.113} C_VEL
LIN {X 0,Y 170.938,Z 498.565,A -85,B 0,C 180,E1 -22999.647,E2 -22999.647} C_VEL
LIN {X 0,Y 169.802,Z 505.965,A -85,B 0,C 180,E1 -23003.86,E2 -23003.86} C_VEL
LIN {X 0,Y 169.248,Z 510.736,A -85,B 0,C 180,E1 -23007.331,E2 -23007.331} C_VEL
LIN {X 0,Y 168.916,Z 514.514,A -85,B 0,C 180,E1 -23010.874,E2 -23010.874} C_VEL
LIN {X 0,Y 169.185,Z 518.039,A -85,B 0,C 180,E1 -23015.458,E2 -23015.458} C_VEL
LIN {X 0,Y 169.744,Z 519.381,A -85,B 0,C 180,E1 -23018.124,E2 -23018.124} C_VEL
LIN {X 0,Y 170.738,Z 520.388,A -85,B 0,C 180,E1 -23021.183,E2 -23021.183} C_VEL
LIN {X 0,Y 171.679,Z 520.703,A -85,B 0,C 180,E1 -23023.35,E2 -23023.35} C_VEL
LIN {X 0,Y 173.448,Z 520.571,A -85,B 0,C 180,E1 -23026.479,E2 -23026.479} C_VEL
LIN {X 0,Y 176.763,Z 519.247,A -85,B 0,C 180,E1 -23030.851,E2 -23030.851} C_VEL
LIN {X 0,Y 178.991,Z 517.851,A -85,B 0,C 180,E1 -23033.237,E2 -23033.237} C_VEL
LIN {X 0,Y 182.993,Z 514.878,A -85,B 0,C 180,E1 -23036.734,E2 -23036.734} C_VEL
LIN {X 0,Y 187.605,Z 510.863,A -85,B 0,C 180,E1 -23040.002,E2 -23040.002} C_VEL
LIN {X 0,Y 192.967,Z 505.529,A -85,B 0,C 180,E1 -23043.134,E2 -23043.134} C_VEL
LIN {X 0,Y 198.767,Z 498.894,A -85,B 0,C 180,E1 -23046.091,E2 -23046.091} C_VEL
LIN {X 0,Y 204.141,Z 492.044,A -85,B 0,C 180,E1 -23048.415,E2 -23048.415} C_VEL
LIN {X 0,Y 204.973,Z 490.687,A -85,B 0,C 180,E1 -23048.878,E2 -23048.878} C_VEL
LIN {X 0,Y 205.942,Z 486.897,A -85,B 0,C 180,E1 -23050.82,E2 -23050.82} C_VEL
LIN {X 0,Y 206.328,Z 482.116,A -85,B 0,C 180,E1 -23053.796,E2 -23053.796} C_VEL
LIN {X 0,Y 206.058,Z 479.452,A -85,B 0,C 180,E1 -23055.836,E2 -23055.836} C_VEL
LIN {X 0,Y 205.706,Z 477.177,A -85,B 0,C 180,E1 -23057.91,E2 -23057.91} C_VEL
LIN {X 0,Y 205.19,Z 475.364,A -85,B 0,C 180,E1 -23060.032,E2 -23060.032} C_VEL
LIN {X 0,Y 204.297,Z 472.932,A -85,B 0,C 180,E1 -23064.383,E2 -23064.383} C_VEL
LIN {X 0,Y 203.798,Z 472.571,A -85,B 0,C 180,E1 -23066.637,E2 -23066.637} C_VEL
LIN {X 0,Y 203.408,Z 473.187,A -85,B 0,C 180,E1 -23071.218,E2 -23071.218} C_VEL
LIN {X 0,Y 203.795,Z 475.498,A -85,B 0,C 180,E1 -23075.894,E2 -23075.894} C_VEL
LIN {X 0,Y 204.05,Z 477.691,A -85,B 0,C 180,E1 -23078.315,E2 -23078.315} C_VEL
LIN {X 0,Y 204.489,Z 480.575,A -85,B 0,C 180,E1 -23080.891,E2 -23080.891} C_VEL
LIN {X 0,Y 204.733,Z 485.095,A -85,B 0,C 180,E1 -23083.885,E2 -23083.885} C_VEL
LIN {X 0,Y 204.7,Z 486.564,A -85,B 0,C 180,E1 -23084.747,E2 -23084.747} C_VEL
LIN {X 0,Y 203.937,Z 490.428,A -85,B 0,C 180,E1 -23086.442,E2 -23086.442} C_VEL
LIN {X 0,Y 201.861,Z 497.342,A -85,B 0,C 180,E1 -23089.259,E2 -23089.259} C_VEL
LIN {X 0,Y 199.036,Z 504.435,A -85,B 0,C 180,E1 -23092.027,E2 -23092.027} C_VEL
LIN {X 0,Y 195.925,Z 510.29,A -85,B 0,C 180,E1 -23094.356,E2 -23094.356} C_VEL
LIN {X 0,Y 189.741,Z 518.126,A -85,B 0,C 180,E1 -23097.525,E2 -23097.525} C_VEL
LIN {X 0,Y 183.268,Z 525.259,A -85,B 0,C 180,E1 -23101.367,E2 -23101.367} C_VEL
LIN {X 0,Y 179.252,Z 529.4,A -85,B 0,C 180,E1 -23104.461,E2 -23104.461} C_VEL
LIN {X 0,Y 177.066,Z 531.698,A -85,B 0,C 180,E1 -23106.624,E2 -23106.624} C_VEL
LIN {X 0,Y 173.292,Z 535.095,A -85,B 0,C 180,E1 -23111.078,E2 -23111.078} C_VEL
LIN {X 0,Y 170.686,Z 537.06,A -85,B 0,C 180,E1 -23115.706,E2 -23115.706} C_VEL
LIN {X 0,Y 169.46,Z 537.63,A -85,B 0,C 180,E1 -23120.46,E2 -23120.46} C_VEL
LIN {X 0,Y 169.279,Z 536.708,A -85,B 0,C 180,E1 -23125.246,E2 -23125.246} C_VEL
LIN {X 0,Y 169.372,Z 535.675,A -85,B 0,C 180,E1 -23127.631,E2 -23127.631} C_VEL
LIN {X 0,Y 169.531,Z 534.226,A -85,B 0,C 180,E1 -23130.009,E2 -23130.009} C_VEL
LIN {X 0,Y 169.542,Z 530.811,A -85,B 0,C 180,E1 -23133.881,E2 -23133.881} C_VEL
LIN {X 0,Y 169.618,Z 526.925,A -85,B 0,C 180,E1 -23137.149,E2 -23137.149} C_VEL
LIN {X 0,Y 170.136,Z 520.444,A -85,B 0,C 180,E1 -23141.324,E2 -23141.324} C_VEL
LIN {X 0,Y 170.464,Z 517.244,A -85,B 0,C 180,E1 -23143.021,E2 -23143.021} C_VEL
LIN {X 0,Y 170.294,Z 513.833,A -85,B 0,C 180,E1 -23144.64,E2 -23144.64} C_VEL
LIN {X 0,Y 168.41,Z 507.677,A -85,B 0,C 180,E1 -23147.203,E2 -23147.203} C_VEL
LIN {X 0,Y 166.781,Z 500.979,A -85,B 0,C 180,E1 -23149.659,E2 -23149.659} C_VEL
LIN {X 0,Y 167.017,Z 496.674,A -85,B 0,C 180,E1 -23151.059,E2 -23151.059} C_VEL
LIN {X 0,Y 168.607,Z 488.953,A -85,B 0,C 180,E1 -23153.257,E2 -23153.257} C_VEL
LIN {X 0,Y 168.218,Z 477.645,A -85,B 0,C 180,E1 -23156.029,E2 -23156.029} C_VEL
LIN {X 0,Y 167.565,Z 465.187,A -85,B 0,C 180,E1 -23158.505,E2 -23158.505} C_VEL
LIN {X 0,Y 166.618,Z 452.269,A -85,B 0,C 180,E1 -23160.588,E2 -23160.588} C_VEL
LIN {X 0,Y 165.433,Z 438.319,A -85,B 0,C 180,E1 -23162.306,E2 -23162.306} C_VEL
LIN {X 0,Y 164.934,Z 433.219,A -85,B 0,C 180,E1 -23162.821,E2 -23162.821} C_VEL
LIN {X 0,Y 165.908,Z 430.293,A -85,B 0,C 180,E1 -23166.401,E2 -23166.401} C_VEL
LIN {X 0,Y 166.164,Z 429.128,A -85,B 0,C 180,E1 -23167.836,E2 -23167.836} C_VEL
LIN {X 0,Y 166.019,Z 427.153,A -85,B 0,C 180,E1 -23170.358,E2 -23170.358} C_VEL
LIN {X 0,Y 165.427,Z 424.578,A -85,B 0,C 180,E1 -23173.758,E2 -23173.758} C_VEL
LIN {X 0,Y 164.54,Z 419.995,A -85,B 0,C 180,E1 -23180.104,E2 -23180.104} C_VEL
LIN {X 0,Y 164.345,Z 420.009,A -85,B 0,C 180,E1 -23186.223,E2 -23186.223} C_VEL
LIN {X 0,Y 164.391,Z 420.009,A -85,B 0,C 180,E1 -23189.132,E2 -23189.132} C_VEL
LIN {X 0,Y 164.415,Z 420.001,A -85,B 0,C 180,E1 -23194.692,E2 -23194.692} C_VEL
LIN {X 0,Y 164.438,Z 419.999,A -85,B 0,C 180,E1 -23200.118,E2 -23200.118} C_VEL
LIN {X 0,Y 164.505,Z 419.995,A -85,B 0,C 180,E1 -23205.145,E2 -23205.145} C_VEL
LIN {X 0,Y 164.786,Z 419.952,A -85,B 0,C 180,E1 -23210.175,E2 -23210.175} C_VEL
LIN {X 0,Y 164.844,Z 419.95,A -85,B 0,C 180,E1 -23212.649,E2 -23212.649} C_VEL
LIN {X 0,Y 165.061,Z 419.919,A -85,B 0,C 180,E1 -23217.558,E2 -23217.558} C_VEL
LIN {X 0,Y 165.303,Z 419.891,A -85,B 0,C 180,E1 -23219.998,E2 -23219.998} C_VEL
LIN {X 0,Y 164.837,Z 419.949,A -85,B 0,C 180,E1 -23227.346,E2 -23227.346} C_VEL
LIN {X 0,Y 164.72,Z 419.967,A -85,B 0,C 180,E1 -23231.053,E2 -23231.053} C_VEL
LIN {X 0,Y 164.454,Z 419.998,A -85,B 0,C 180,E1 -23237.404,E2 -23237.404} C_VEL
LIN {X 0,Y 164.368,Z 420.007,A -85,B 0,C 180,E1 -23242.63,E2 -23242.63} C_VEL
LIN {X 0,Y 164.4,Z 420.005,A -85,B 0,C 180,E1 -23246.121,E2 -23246.121} C_VEL
LIN {X 0,Y 164.386,Z 420.003,A -85,B 0,C 180,E1 -23251.22,E2 -23251.22} C_VEL
LIN {X 0,Y 164.307,Z 420.018,A -85,B 0,C 180,E1 -23256.783,E2 -23256.783} C_VEL
LIN {X 0,Y 164.303,Z 420.014,A -85,B 0,C 180,E1 -23259.91,E2 -23259.91} C_VEL
LIN {X 0,Y 164.291,Z 420.019,A -85,B 0,C 180,E1 -23263.335,E2 -23263.335} C_VEL
LIN {X 0,Y 164.271,Z 420.02,A -85,B 0,C 180,E1 -23266.791,E2 -23266.791} C_VEL
LIN {X 0,Y 164.299,Z 420.017,A -85,B 0,C 180,E1 -23270.347,E2 -23270.347} C_VEL
LIN {X 0,Y 164.333,Z 420.012,A -85,B 0,C 180,E1 -23276.213,E2 -23276.213} C_VEL
LIN {X 0,Y 164.396,Z 420.005,A -85,B 0,C 180,E1 -23279.126,E2 -23279.126} C_VEL
LIN {X 0,Y 164.421,Z 419.999,A -85,B 0,C 180,E1 -23284.686,E2 -23284.686} C_VEL
LIN {X 0,Y 164.487,Z 419.996,A -85,B 0,C 180,E1 -23290.042,E2 -23290.042} C_VEL
LIN {X 0,Y 164.524,Z 419.988,A -85,B 0,C 180,E1 -23295.14,E2 -23295.14} C_VEL
LIN {X 0,Y 164.766,Z 419.96,A -85,B 0,C 180,E1 -23300.168,E2 -23300.168} C_VEL
LIN {X 0,Y 164.828,Z 419.95,A -85,B 0,C 180,E1 -23302.642,E2 -23302.642} C_VEL
LIN {X 0,Y 165.042,Z 419.925,A -85,B 0,C 180,E1 -23307.551,E2 -23307.551} C_VEL
LIN {X 0,Y 165.289,Z 419.892,A -85,B 0,C 180,E1 -23309.991,E2 -23309.991} C_VEL
LIN {X 0,Y 164.767,Z 419.96,A -85,B 0,C 180,E1 -23314.885,E2 -23314.885} C_VEL
LIN {X 0,Y 164.852,Z 419.947,A -85,B 0,C 180,E1 -23317.339,E2 -23317.339} C_VEL
LIN {X 0,Y 164.769,Z 419.958,A -85,B 0,C 180,E1 -23321.189,E2 -23321.189} C_VEL
LIN {X 0,Y 164.49,Z 419.989,A -85,B 0,C 180,E1 -23327.393,E2 -23327.393} C_VEL
LIN {X 0,Y 164.456,Z 420,A -85,B 0,C 180,E1 -23329.981,E2 -23329.981} C_VEL
LIN {X 0,Y 164.155,Z 420.038,A -85,B 0,C 180,E1 -23335.969,E2 -23335.969} C_VEL
LIN {X 0,Y 163.895,Z 420.211,A -85,B 0,C 180,E1 -23339.712,E2 -23339.712} C_VEL
LIN {X 0,Y 167.486,Z 433.097,A -85,B 0,C 180,E1 -23341.624,E2 -23341.624} C_VEL
LIN {X 0,Y 170.038,Z 446.132,A -85,B 0,C 180,E1 -23343.906,E2 -23343.906} C_VEL
LIN {X 0,Y 171.732,Z 456.396,A -85,B 0,C 180,E1 -23346.023,E2 -23346.023} C_VEL
LIN {X 0,Y 171.296,Z 460.417,A -85,B 0,C 180,E1 -23346.869,E2 -23346.869} C_VEL
LIN {X 0,Y 169.245,Z 470.945,A -85,B 0,C 180,E1 -23349.357,E2 -23349.357} C_VEL
LIN {X 0,Y 167.303,Z 480.694,A -85,B 0,C 180,E1 -23352.218,E2 -23352.218} C_VEL
LIN {X 0,Y 165.249,Z 490.854,A -85,B 0,C 180,E1 -23355.957,E2 -23355.957} C_VEL
LIN {X 0,Y 163.961,Z 497.91,A -85,B 0,C 180,E1 -23359.184,E2 -23359.184} C_VEL
LIN {X 0,Y 162.926,Z 504.416,A -85,B 0,C 180,E1 -23362.853,E2 -23362.853} C_VEL
LIN {X 0,Y 162.174,Z 510.442,A -85,B 0,C 180,E1 -23367.203,E2 -23367.203} C_VEL
LIN {X 0,Y 161.82,Z 514.91,A -85,B 0,C 180,E1 -23371.465,E2 -23371.465} C_VEL
LIN {X 0,Y 162.09,Z 518.021,A -85,B 0,C 180,E1 -23375.553,E2 -23375.553} C_VEL
LIN {X 0,Y 163.525,Z 520.509,A -85,B 0,C 180,E1 -23380.967,E2 -23380.967} C_VEL
LIN {X 0,Y 165.489,Z 521.2,A -85,B 0,C 180,E1 -23385.24,E2 -23385.24} C_VEL
LIN {X 0,Y 167.15,Z 521.058,A -85,B 0,C 180,E1 -23387.866,E2 -23387.866} C_VEL
LIN {X 0,Y 170.35,Z 519.934,A -85,B 0,C 180,E1 -23391.877,E2 -23391.877} C_VEL
LIN {X 0,Y 173.878,Z 517.975,A -85,B 0,C 180,E1 -23395.365,E2 -23395.365} C_VEL
LIN {X 0,Y 178.315,Z 514.886,A -85,B 0,C 180,E1 -23398.873,E2 -23398.873} C_VEL
LIN {X 0,Y 183.436,Z 510.648,A -85,B 0,C 180,E1 -23402.198,E2 -23402.198} C_VEL
LIN {X 0,Y 189.194,Z 505.21,A -85,B 0,C 180,E1 -23405.332,E2 -23405.332} C_VEL
LIN {X 0,Y 195.513,Z 498.295,A -85,B 0,C 180,E1 -23408.269,E2 -23408.269} C_VEL
LIN {X 0,Y 198.924,Z 494.175,A -85,B 0,C 180,E1 -23409.663,E2 -23409.663} C_VEL
LIN {X 0,Y 199.597,Z 493.059,A -85,B 0,C 180,E1 -23410.142,E2 -23410.142} C_VEL
LIN {X 0,Y 200.633,Z 489.69,A -85,B 0,C 180,E1 -23412.134,E2 -23412.134} C_VEL
LIN {X 0,Y 201.143,Z 485.347,A -85,B 0,C 180,E1 -23415.195,E2 -23415.195} C_VEL
LIN {X 0,Y 200.821,Z 482.127,A -85,B 0,C 180,E1 -23418.361,E2 -23418.361} C_VEL
LIN {X 0,Y 200.463,Z 480.514,A -85,B 0,C 180,E1 -23420.525,E2 -23420.525} C_VEL
LIN {X 0,Y 199.947,Z 478.732,A -85,B 0,C 180,E1 -23423.975,E2 -23423.975} C_VEL
LIN {X 0,Y 199.383,Z 478.264,A -85,B 0,C 180,E1 -23427.275,E2 -23427.275} C_VEL
LIN {X 0,Y 199.137,Z 478.494,A -85,B 0,C 180,E1 -23429.612,E2 -23429.612} C_VEL
LIN {X 0,Y 199.081,Z 479.225,A -85,B 0,C 180,E1 -23432.103,E2 -23432.103} C_VEL
LIN {X 0,Y 199.378,Z 481.134,A -85,B 0,C 180,E1 -23435.847,E2 -23435.847} C_VEL
LIN {X 0,Y 199.463,Z 482.563,A -85,B 0,C 180,E1 -23437.581,E2 -23437.581} C_VEL
LIN {X 0,Y 199.671,Z 486.224,A -85,B 0,C 180,E1 -23440.938,E2 -23440.938} C_VEL
LIN {X 0,Y 199.651,Z 489.629,A -85,B 0,C 180,E1 -23443.327,E2 -23443.327} C_VEL
LIN {X 0,Y 199.102,Z 492.506,A -85,B 0,C 180,E1 -23444.91,E2 -23444.91} C_VEL
LIN {X 0,Y 196.596,Z 499.548,A -85,B 0,C 180,E1 -23447.992,E2 -23447.992} C_VEL
LIN {X 0,Y 193.044,Z 507.043,A -85,B 0,C 180,E1 -23451.179,E2 -23451.179} C_VEL
LIN {X 0,Y 190.284,Z 511.599,A -85,B 0,C 180,E1 -23453.128,E2 -23453.128} C_VEL
LIN {X 0,Y 183.854,Z 519.035,A -85,B 0,C 180,E1 -23456.35,E2 -23456.35} C_VEL
LIN {X 0,Y 178.707,Z 524.267,A -85,B 0,C 180,E1 -23459.264,E2 -23459.264} C_VEL
LIN {X 0,Y 174.213,Z 528.514,A -85,B 0,C 180,E1 -23462.37,E2 -23462.37} C_VEL
LIN {X 0,Y 170.567,Z 531.845,A -85,B 0,C 180,E1 -23465.677,E2 -23465.677} C_VEL
LIN {X 0,Y 166.584,Z 535.011,A -85,B 0,C 180,E1 -23470.285,E2 -23470.285} C_VEL
LIN {X 0,Y 163.775,Z 536.762,A -85,B 0,C 180,E1 -23475.09,E2 -23475.09} C_VEL
LIN {X 0,Y 162.449,Z 537.072,A -85,B 0,C 180,E1 -23480.044,E2 -23480.044} C_VEL
LIN {X 0,Y 162.22,Z 535.91,A -85,B 0,C 180,E1 -23485.192,E2 -23485.192} C_VEL
LIN {X 0,Y 162.316,Z 534.846,A -85,B 0,C 180,E1 -23487.528,E2 -23487.528} C_VEL
LIN {X 0,Y 162.448,Z 532.321,A -85,B 0,C 180,E1 -23491.249,E2 -23491.249} C_VEL
LIN {X 0,Y 162.546,Z 528.719,A -85,B 0,C 180,E1 -23494.97,E2 -23494.97} C_VEL
LIN {X 0,Y 162.677,Z 523.896,A -85,B 0,C 180,E1 -23498.706,E2 -23498.706} C_VEL
LIN {X 0,Y 163.25,Z 517.776,A -85,B 0,C 180,E1 -23502.439,E2 -23502.439} C_VEL
LIN {X 0,Y 164.519,Z 510.136,A -85,B 0,C 180,E1 -23506.13,E2 -23506.13} C_VEL
LIN {X 0,Y 166.156,Z 500.603,A -85,B 0,C 180,E1 -23509.787,E2 -23509.787} C_VEL
LIN {X 0,Y 167.017,Z 496.674,A -85,B 0,C 180,E1 -23511.059,E2 -23511.059} C_VEL
LIN {X 0,Y 167.239,Z 493.737,A -85,B 0,C 180,E1 -23511.95,E2 -23511.95} C_VEL
LIN {X 0,Y 166.394,Z 489.286,A -85,B 0,C 180,E1 -23513.264,E2 -23513.264} C_VEL
LIN {X 0,Y 164.737,Z 484.842,A -85,B 0,C 180,E1 -23514.528,E2 -23514.528} C_VEL
LIN {X 0,Y 162.26,Z 478.651,A -85,B 0,C 180,E1 -23516.167,E2 -23516.167} C_VEL
LIN {X 0,Y 161.034,Z 473.693,A -85,B 0,C 180,E1 -23517.327,E2 -23517.327} C_VEL
LIN {X 0,Y 160.871,Z 471.959,A -85,B 0,C 180,E1 -23517.692,E2 -23517.692} C_VEL
LIN {X 0,Y 160.174,Z 459.099,A -85,B 0,C 180,E1 -23520.13,E2 -23520.13} C_VEL
LIN {X 0,Y 159.229,Z 446.195,A -85,B 0,C 180,E1 -23522.093,E2 -23522.093} C_VEL
LIN {X 0,Y 158.065,Z 432.794,A -85,B 0,C 180,E1 -23523.668,E2 -23523.668} C_VEL
LIN {X 0,Y 158.944,Z 430.006,A -85,B 0,C 180,E1 -23527.256,E2 -23527.256} C_VEL
LIN {X 0,Y 159.007,Z 428.193,A -85,B 0,C 180,E1 -23529.663,E2 -23529.663} C_VEL
LIN {X 0,Y 158.166,Z 424.55,A -85,B 0,C 180,E1 -23534.685,E2 -23534.685} C_VEL
LIN {X 0,Y 157.473,Z 420.868,A -85,B 0,C 180,E1 -23540.315,E2 -23540.315} C_VEL
LIN {X 0,Y 157.31,Z 420.885,A -85,B 0,C 180,E1 -23544.491,E2 -23544.491} C_VEL
LIN {X 0,Y 157.304,Z 420.889,A -85,B 0,C 180,E1 -23548.105,E2 -23548.105} C_VEL
LIN {X 0,Y 157.331,Z 420.883,A -85,B 0,C 180,E1 -23553.465,E2 -23553.465} C_VEL
LIN {X 0,Y 157.381,Z 420.878,A -85,B 0,C 180,E1 -23559.703,E2 -23559.703} C_VEL
LIN {X 0,Y 157.437,Z 420.872,A -85,B 0,C 180,E1 -23564.462,E2 -23564.462} C_VEL
LIN {X 0,Y 157.708,Z 420.834,A -85,B 0,C 180,E1 -23569.73,E2 -23569.73} C_VEL
LIN {X 0,Y 157.782,Z 420.828,A -85,B 0,C 180,E1 -23572.319,E2 -23572.319} C_VEL
LIN {X 0,Y 158.264,Z 420.767,A -85,B 0,C 180,E1 -23579.998,E2 -23579.998} C_VEL
LIN {X 0,Y 157.776,Z 420.827,A -85,B 0,C 180,E1 -23587.677,E2 -23587.677} C_VEL
LIN {X 0,Y 157.651,Z 420.847,A -85,B 0,C 180,E1 -23591.221,E2 -23591.221} C_VEL
LIN {X 0,Y 157.433,Z 420.869,A -85,B 0,C 180,E1 -23595.534,E2 -23595.534} C_VEL
LIN {X 0,Y 157.328,Z 420.886,A -85,B 0,C 180,E1 -23600.936,E2 -23600.936} C_VEL
LIN {X 0,Y 157.326,Z 420.888,A -85,B 0,C 180,E1 -23606.675,E2 -23606.675} C_VEL
LIN {X 0,Y 157.288,Z 420.887,A -85,B 0,C 180,E1 -23612.422,E2 -23612.422} C_VEL
LIN {X 0,Y 157.281,Z 420.894,A -85,B 0,C 180,E1 -23616.442,E2 -23616.442} C_VEL
LIN {X 0,Y 157.204,Z 420.9,A -85,B 0,C 180,E1 -23622.11,E2 -23622.11} C_VEL
LIN {X 0,Y 157.2,Z 420.899,A -85,B 0,C 180,E1 -23627.875,E2 -23627.875} C_VEL
LIN {X 0,Y 157.267,Z 420.894,A -85,B 0,C 180,E1 -23633.547,E2 -23633.547} C_VEL
LIN {X 0,Y 157.299,Z 420.887,A -85,B 0,C 180,E1 -23638.088,E2 -23638.088} C_VEL
LIN {X 0,Y 157.327,Z 420.885,A -85,B 0,C 180,E1 -23643.457,E2 -23643.457} C_VEL
LIN {X 0,Y 157.396,Z 420.878,A -85,B 0,C 180,E1 -23649.658,E2 -23649.658} C_VEL
LIN {X 0,Y 157.454,Z 420.868,A -85,B 0,C 180,E1 -23654.457,E2 -23654.457} C_VEL
LIN {X 0,Y 157.688,Z 420.842,A -85,B 0,C 180,E1 -23659.721,E2 -23659.721} C_VEL
LIN {X 0,Y 157.765,Z 420.829,A -85,B 0,C 180,E1 -23662.311,E2 -23662.311} C_VEL
LIN {X 0,Y 158.251,Z 420.768,A -85,B 0,C 180,E1 -23669.991,E2 -23669.991} C_VEL
LIN {X 0,Y 157.815,Z 420.824,A -85,B 0,C 180,E1 -23677.668,E2 -23677.668} C_VEL
LIN {X 0,Y 157.694,Z 420.84,A -85,B 0,C 180,E1 -23681.353,E2 -23681.353} C_VEL
LIN {X 0,Y 157.464,Z 420.868,A -85,B 0,C 180,E1 -23685.523,E2 -23685.523} C_VEL
LIN {X 0,Y 157.311,Z 420.889,A -85,B 0,C 180,E1 -23690.93,E2 -23690.93} C_VEL
LIN {X 0,Y 157.196,Z 420.903,A -85,B 0,C 180,E1 -23693.716,E2 -23693.716} C_VEL
LIN {X 0,Y 156.862,Z 420.945,A -85,B 0,C 180,E1 -23698.964,E2 -23698.964} C_VEL
LIN {X 0,Y 160.58,Z 434.428,A -85,B 0,C 180,E1 -23701.086,E2 -23701.086} C_VEL
LIN {X 0,Y 162.954,Z 446.286,A -85,B 0,C 180,E1 -23703.255,E2 -23703.255} C_VEL
LIN {X 0,Y 164.67,Z 456.616,A -85,B 0,C 180,E1 -23705.479,E2 -23705.479} C_VEL
LIN {X 0,Y 164.504,Z 459.735,A -85,B 0,C 180,E1 -23706.168,E2 -23706.168} C_VEL
LIN {X 0,Y 162.14,Z 471.724,A -85,B 0,C 180,E1 -23709.1,E2 -23709.1} C_VEL
LIN {X 0,Y 160.064,Z 481.655,A -85,B 0,C 180,E1 -23712.192,E2 -23712.192} C_VEL
LIN {X 0,Y 158.125,Z 491.189,A -85,B 0,C 180,E1 -23715.894,E2 -23715.894} C_VEL
LIN {X 0,Y 156.672,Z 499.011,A -85,B 0,C 180,E1 -23719.676,E2 -23719.676} C_VEL
LIN {X 0,Y 155.589,Z 506.125,A -85,B 0,C 180,E1 -23724.043,E2 -23724.043} C_VEL
LIN {X 0,Y 154.919,Z 511.699,A -85,B 0,C 180,E1 -23728.431,E2 -23728.431} C_VEL
LIN {X 0,Y 154.752,Z 516.059,A -85,B 0,C 180,E1 -23732.993,E2 -23732.993} C_VEL
LIN {X 0,Y 155.037,Z 518.134,A -85,B 0,C 180,E1 -23735.925,E2 -23735.925} C_VEL
LIN {X 0,Y 156.29,Z 520.529,A -85,B 0,C 180,E1 -23740.757,E2 -23740.757} C_VEL
LIN {X 0,Y 157.904,Z 521.497,A -85,B 0,C 180,E1 -23744.514,E2 -23744.514} C_VEL
LIN {X 0,Y 159.487,Z 521.701,A -85,B 0,C 180,E1 -23747.274,E2 -23747.274} C_VEL
LIN {X 0,Y 163.166,Z 520.968,A -85,B 0,C 180,E1 -23752.088,E2 -23752.088} C_VEL
LIN {X 0,Y 166.171,Z 519.664,A -85,B 0,C 180,E1 -23755.15,E2 -23755.15} C_VEL
LIN {X 0,Y 170.559,Z 517.139,A -85,B 0,C 180,E1 -23758.822,E2 -23758.822} C_VEL
LIN {X 0,Y 175.814,Z 513.499,A -85,B 0,C 180,E1 -23762.331,E2 -23762.331} C_VEL
LIN {X 0,Y 181.617,Z 508.75,A -85,B 0,C 180,E1 -23765.554,E2 -23765.554} C_VEL
LIN {X 0,Y 187.997,Z 502.66,A -85,B 0,C 180,E1 -23768.602,E2 -23768.602} C_VEL
LIN {X 0,Y 193.072,Z 497.253,A -85,B 0,C 180,E1 -23770.685,E2 -23770.685} C_VEL
LIN {X 0,Y 194.309,Z 495.492,A -85,B 0,C 180,E1 -23771.475,E2 -23771.475} C_VEL
LIN {X 0,Y 195.399,Z 492.019,A -85,B 0,C 180,E1 -23773.843,E2 -23773.843} C_VEL
LIN {X 0,Y 195.851,Z 489.848,A -85,B 0,C 180,E1 -23775.614,E2 -23775.614} C_VEL
LIN {X 0,Y 195.771,Z 486.899,A -85,B 0,C 180,E1 -23778.852,E2 -23778.852} C_VEL
LIN {X 0,Y 195.537,Z 485.446,A -85,B 0,C 180,E1 -23781.066,E2 -23781.066} C_VEL
LIN {X 0,Y 195.331,Z 484.377,A -85,B 0,C 180,E1 -23783.316,E2 -23783.316} C_VEL
LIN {X 0,Y 195.016,Z 483.763,A -85,B 0,C 180,E1 -23785.738,E2 -23785.738} C_VEL
LIN {X 0,Y 194.543,Z 484.018,A -85,B 0,C 180,E1 -23789.905,E2 -23789.905} C_VEL
LIN {X 0,Y 194.531,Z 485.394,A -85,B 0,C 180,E1 -23793.821,E2 -23793.821} C_VEL
LIN {X 0,Y 194.65,Z 486.22,A -85,B 0,C 180,E1 -23795.29,E2 -23795.29} C_VEL
LIN {X 0,Y 194.632,Z 488.279,A -85,B 0,C 180,E1 -23797.871,E2 -23797.871} C_VEL
LIN {X 0,Y 194.622,Z 491.234,A -85,B 0,C 180,E1 -23800.696,E2 -23800.696} C_VEL
LIN {X 0,Y 194.174,Z 495.039,A -85,B 0,C 180,E1 -23803.45,E2 -23803.45} C_VEL
LIN {X 0,Y 192.032,Z 500.181,A -85,B 0,C 180,E1 -23805.956,E2 -23805.956} C_VEL
LIN {X 0,Y 189.697,Z 505.007,A -85,B 0,C 180,E1 -23808.186,E2 -23808.186} C_VEL
